(* IEC 61131-3 sources: scada_scout/plc_programs, 162 files *)

(* ---- PRG_GBCUPM01.st ---- *)
(* ========================================================================
   PLC PROGRAM: PRG_GBCUPM01
   IED: GBCUPM01
   Device: GBCUPM01
   Generated: 2026-02-05 10:55:39

   This program runs cyclically (default 100ms) and has access to all
   data points of the associated IEC 61850 device. Users can add custom
   logic in the designated sections below.
   ======================================================================== *)

PROGRAM PRG_GBCUPM01
VAR
    (* ====== System Variables ====== *)
    cycle_count: UDINT := 0;           (* Increments each scan cycle *)
    first_scan: BOOL := TRUE;          (* TRUE only on first execution *)
    scan_time_ms: REAL := 0.0;         (* Last scan time in milliseconds *)

    (* ====== IED Connection Status ====== *)
    ied_connected: BOOL := FALSE;      (* TRUE when IED server is running *)
    ied_name: STRING := 'GBCUPM01';
    device_name: STRING := 'GBCUPM01';

    (* ====== Logical Devices ====== *)
    (* Available LDs: AnUn_ArcProtInput1, Application, BinIO, BinIO_BinaryInputs, BinIO_BinaryOutputs, CB1, CB1_Fundamental, Ds1, Ds2, Mod1, Mod1_Channel1, Mod2, Mod2_Channel1, Mod3, Mod3_Channel1, PowS, PowS_MeasPointI3ph1, PowS_MeasPointV3ph1, Rec, Rec_FaultRecorder, VI3p1, VI3p1_5051NOCgndB1, VI3p1_5051OC3phase1, VI3p1_ArcProtection1, VI3p1_Energy, VI3p1_FundSymComp, VI3p1_OperationalValues, VI3p1_ProcessMonitor, CB2, CB2_Fundamental, CB3, CB3_Fundamental, ComSupervision, ComSupervision_GOOSE *)

    (* ====== User Variables ====== *)
    (* Add your custom variables here *)
    (* Example:
    timer1: TON;
    counter: INT := 0;
    status_word: WORD;
    *)

END_VAR

(* ======================================================================
   INITIALIZATION SECTION
   Runs once on first scan. Use for setup and initialization.
   ====================================================================== *)
IF first_scan THEN
    (* Initialize user variables here *)
    cycle_count := 0;

    (* Log program start *)
    (* SCADA_LOG('INFO', CONCAT('PLC Program started: ', device_name)); *)

    first_scan := FALSE;
END_IF;

(* ======================================================================
   MAIN CYCLIC EXECUTION
   This section runs continuously every scan cycle (default 100ms).
   ====================================================================== *)

(* Increment cycle counter *)
cycle_count := cycle_count + 1;

(* ====== USER LOGIC SECTION 1: Pre-Processing ====== *)
(* Add logic that should run before main processing *)
(* Example:
IF ied_connected THEN
    (* Read IED data points *)
    (* status_word := READ_IED_DATA(device_name, 'LD0/MMXU1$MX$TotW$mag'); *)
END_IF;
*)

(* ====== USER LOGIC SECTION 2: Main Processing ====== *)
(* Add your main control logic here *)
(* Example:
IF counter > 100 THEN
    counter := 0;
    (* Perform periodic action *)
END_IF;
counter := counter + 1;
*)

(* ====== USER LOGIC SECTION 3: Post-Processing ====== *)
(* Add logic for outputs, writes, and cleanup *)
(* Example:
IF ied_connected THEN
    (* Write control commands to IED *)
    (* WRITE_IED_CONTROL(device_name, 'LD0/CSWI1$CO$Pos', TRUE); *)
END_IF;
*)

(* ====== Built-in Functions Available ====== *)
(*
   READ_IED_DATA(device: STRING, ref: STRING): ANY
       - Read data from IED object reference
       - Example: READ_IED_DATA('MyIED', 'LD0/MMXU1$MX$TotW$mag')

   WRITE_IED_DATA(device: STRING, ref: STRING, value: ANY): BOOL
       - Write data to IED object reference
       - Returns TRUE on success

   WRITE_IED_CONTROL(device: STRING, ref: STRING, value: ANY): BOOL
       - Send control command to IED
       - Returns TRUE on success

   SCADA_LOG(level: STRING, message: STRING)
       - Log message to event log
       - Levels: 'INFO', 'WARNING', 'ERROR'

   GET_DEVICE_STATUS(device: STRING): BOOL
       - Check if device is connected
*)

END_PROGRAM

(* ---- PRG_GPS01ECB01.st ---- *)
(* ========================================================================
   PLC PROGRAM: PRG_GPS01ECB01
   IED: GPS01ECB01
   Device: GPS01ECB01
   Generated: 2026-02-05 10:51:13

   This program runs cyclically (default 100ms) and has access to all
   data points of the associated IEC 61850 device. Users can add custom
   logic in the designated sections below.
   ======================================================================== *)

PROGRAM PRG_GPS01ECB01
VAR
    (* ====== System Variables ====== *)
    cycle_count: UDINT := 0;           (* Increments each scan cycle *)
    first_scan: BOOL := TRUE;          (* TRUE only on first execution *)
    scan_time_ms: REAL := 0.0;         (* Last scan time in milliseconds *)

    (* ====== IED Connection Status ====== *)
    ied_connected: BOOL := FALSE;      (* TRUE when IED server is running *)
    ied_name: STRING := 'GPS01ECB01';
    device_name: STRING := 'GPS01ECB01';

    (* ====== Logical Devices ====== *)
    (* Available LDs: AnUn_ArcProtInput1, Application, BinIO, BinIO_BinaryInputs, BinIO_BinaryOutputs, CB1, CB1_Fundamental, Ds1, Ds2, Mod1, Mod1_Channel1, Mod2, Mod2_Channel1, Mod3, Mod3_Channel1, PowS, PowS_MeasPointI3ph1, PowS_MeasPointV3ph1, Rec, Rec_FaultRecorder, VI3p1, VI3p1_5051NOCgndB1, VI3p1_5051OC3phase1, VI3p1_67DirOC3phB1, VI3p1_67NDirOCgndB1, VI3p1_ArcProtection1, VI3p1_Energy, VI3p1_FundSymComp, VI3p1_OperationalValues, VI3p1_ProcessMonitor, VI3p1_ExternalTrip1, VI3p1_ExternalTrip2, PowS_MeasPointI1ph1, VI1p1, VI1p1_50N51NOC1phB1, VI1p1_Fundamental, ComSupervision, ComSupervision_GOOSE *)

    (* ====== User Variables ====== *)
    (* Add your custom variables here *)
    (* Example:
    timer1: TON;
    counter: INT := 0;
    status_word: WORD;
    *)

END_VAR

(* ======================================================================
   INITIALIZATION SECTION
   Runs once on first scan. Use for setup and initialization.
   ====================================================================== *)
IF first_scan THEN
    (* Initialize user variables here *)
    cycle_count := 0;

    (* Log program start *)
    (* SCADA_LOG('INFO', CONCAT('PLC Program started: ', device_name)); *)

    first_scan := FALSE;
END_IF;

(* ======================================================================
   MAIN CYCLIC EXECUTION
   This section runs continuously every scan cycle (default 100ms).
   ====================================================================== *)

(* Increment cycle counter *)
cycle_count := cycle_count + 1;

(* ====== USER LOGIC SECTION 1: Pre-Processing ====== *)
(* Add logic that should run before main processing *)
(* Example:
IF ied_connected THEN
    (* Read IED data points *)
    (* status_word := READ_IED_DATA(device_name, 'LD0/MMXU1$MX$TotW$mag'); *)
END_IF;
*)

(* ====== USER LOGIC SECTION 2: Main Processing ====== *)
(* Add your main control logic here *)
(* Example:
IF counter > 100 THEN
    counter := 0;
    (* Perform periodic action *)
END_IF;
counter := counter + 1;
*)

(* ====== USER LOGIC SECTION 3: Post-Processing ====== *)
(* Add logic for outputs, writes, and cleanup *)
(* Example:
IF ied_connected THEN
    (* Write control commands to IED *)
    (* WRITE_IED_CONTROL(device_name, 'LD0/CSWI1$CO$Pos', TRUE); *)
END_IF;
*)

(* ====== Built-in Functions Available ====== *)
(*
   READ_IED_DATA(device: STRING, ref: STRING): ANY
       - Read data from IED object reference
       - Example: READ_IED_DATA('MyIED', 'LD0/MMXU1$MX$TotW$mag')

   WRITE_IED_DATA(device: STRING, ref: STRING, value: ANY): BOOL
       - Write data to IED object reference
       - Returns TRUE on success

   WRITE_IED_CONTROL(device: STRING, ref: STRING, value: ANY): BOOL
       - Send control command to IED
       - Returns TRUE on success

   SCADA_LOG(level: STRING, message: STRING)
       - Log message to event log
       - Levels: 'INFO', 'WARNING', 'ERROR'

   GET_DEVICE_STATUS(device: STRING): BOOL
       - Check if device is connected
*)

END_PROGRAM

(* ---- PRG_GPS01FCB01.st ---- *)
(* ========================================================================
   PLC PROGRAM: PRG_GPS01FCB01
   IED: GPS01FCB01
   Device: GPS01FCB01
   Generated: 2026-02-05 10:51:08

   This program runs cyclically (default 100ms) and has access to all
   data points of the associated IEC 61850 device. Users can add custom
   logic in the designated sections below.
   ======================================================================== *)

PROGRAM PRG_GPS01FCB01
VAR
    (* ====== System Variables ====== *)
    cycle_count: UDINT := 0;           (* Increments each scan cycle *)
    first_scan: BOOL := TRUE;          (* TRUE only on first execution *)
    scan_time_ms: REAL := 0.0;         (* Last scan time in milliseconds *)

    (* ====== IED Connection Status ====== *)
    ied_connected: BOOL := FALSE;      (* TRUE when IED server is running *)
    ied_name: STRING := 'GPS01FCB01';
    device_name: STRING := 'GPS01FCB01';

    (* ====== Logical Devices ====== *)
    (* Available LDs: AnUn_ArcProtInput1, Application, BinIO, BinIO_BinaryInputs, BinIO_BinaryOutputs, CB1, CB1_Fundamental, Ds1, Ds2, Mod1, Mod1_Channel1, Mod2, Mod2_Channel1, Mod3, Mod3_Channel1, PowS, PowS_MeasPointI3ph1, PowS_MeasPointV1ph1, PowS_MeasPointV3ph1, Rec, Rec_FaultRecorder, VI1p1, VI1p1_Fundamental, VI3p1, VI3p1_5051NOCgndB1, VI3p1_5051OC3phase1, VI3p1_67DirOC3phB1, VI3p1_67NDirOCgndB1, VI3p1_ArcProtection1, VI3p1_Energy, VI3p1_FundSymComp, VI3p1_OperationalValues, VI3p1_ProcessMonitor, VI3p1_ExternalTrip1, VI3p1_ExternalTrip2, ComSupervision, ComSupervision_GOOSE *)

    (* ====== User Variables ====== *)
    (* Add your custom variables here *)
    (* Example:
    timer1: TON;
    counter: INT := 0;
    status_word: WORD;
    *)

END_VAR

(* ======================================================================
   INITIALIZATION SECTION
   Runs once on first scan. Use for setup and initialization.
   ====================================================================== *)
IF first_scan THEN
    (* Initialize user variables here *)
    cycle_count := 0;

    (* Log program start *)
    (* SCADA_LOG('INFO', CONCAT('PLC Program started: ', device_name)); *)

    first_scan := FALSE;
END_IF;

(* ======================================================================
   MAIN CYCLIC EXECUTION
   This section runs continuously every scan cycle (default 100ms).
   ====================================================================== *)

(* Increment cycle counter *)
cycle_count := cycle_count + 1;

(* ====== USER LOGIC SECTION 1: Pre-Processing ====== *)
(* Add logic that should run before main processing *)
(* Example:
IF ied_connected THEN
    (* Read IED data points *)
    (* status_word := READ_IED_DATA(device_name, 'LD0/MMXU1$MX$TotW$mag'); *)
END_IF;
*)

(* ====== USER LOGIC SECTION 2: Main Processing ====== *)
(* Add your main control logic here *)
(* Example:
IF counter > 100 THEN
    counter := 0;
    (* Perform periodic action *)
END_IF;
counter := counter + 1;
*)

(* ====== USER LOGIC SECTION 3: Post-Processing ====== *)
(* Add logic for outputs, writes, and cleanup *)
(* Example:
IF ied_connected THEN
    (* Write control commands to IED *)
    (* WRITE_IED_CONTROL(device_name, 'LD0/CSWI1$CO$Pos', TRUE); *)
END_IF;
*)

(* ====== Built-in Functions Available ====== *)
(*
   READ_IED_DATA(device: STRING, ref: STRING): ANY
       - Read data from IED object reference
       - Example: READ_IED_DATA('MyIED', 'LD0/MMXU1$MX$TotW$mag')

   WRITE_IED_DATA(device: STRING, ref: STRING, value: ANY): BOOL
       - Write data to IED object reference
       - Returns TRUE on success

   WRITE_IED_CONTROL(device: STRING, ref: STRING, value: ANY): BOOL
       - Send control command to IED
       - Returns TRUE on success

   SCADA_LOG(level: STRING, message: STRING)
       - Log message to event log
       - Levels: 'INFO', 'WARNING', 'ERROR'

   GET_DEVICE_STATUS(device: STRING): BOOL
       - Check if device is connected
*)

END_PROGRAM

(* ---- PRG_GPS01FCB02.st ---- *)
(* ========================================================================
   PLC PROGRAM: PRG_GPS01FCB02
   IED: GPS01FCB02
   Device: GPS01FCB02
   Generated: 2026-02-05 10:51:10

   This program runs cyclically (default 100ms) and has access to all
   data points of the associated IEC 61850 device. Users can add custom
   logic in the designated sections below.
   ======================================================================== *)

PROGRAM PRG_GPS01FCB02
VAR
    (* ====== System Variables ====== *)
    cycle_count: UDINT := 0;           (* Increments each scan cycle *)
    first_scan: BOOL := TRUE;          (* TRUE only on first execution *)
    scan_time_ms: REAL := 0.0;         (* Last scan time in milliseconds *)

    (* ====== IED Connection Status ====== *)
    ied_connected: BOOL := FALSE;      (* TRUE when IED server is running *)
    ied_name: STRING := 'GPS01FCB02';
    device_name: STRING := 'GPS01FCB02';

    (* ====== Logical Devices ====== *)
    (* Available LDs: AnUn_ArcProtInput1, Application, BinIO, BinIO_BinaryInputs, BinIO_BinaryOutputs, CB1, CB1_Fundamental, Ds1, Ds2, Mod1, Mod1_Channel1, Mod2, Mod2_Channel1, Mod3, Mod3_Channel1, PowS, PowS_MeasPointI3ph1, PowS_MeasPointV1ph1, PowS_MeasPointV3ph1, Rec, Rec_FaultRecorder, VI1p1, VI1p1_Fundamental, VI3p1, VI3p1_5051NOCgndB1, VI3p1_5051OC3phase1, VI3p1_67DirOC3phB1, VI3p1_67NDirOCgndB1, VI3p1_ArcProtection1, VI3p1_Energy, VI3p1_FundSymComp, VI3p1_OperationalValues, VI3p1_ProcessMonitor, VI3p1_ExternalTrip1, VI3p1_ExternalTrip2, ComSupervision, ComSupervision_GOOSE *)

    (* ====== User Variables ====== *)
    (* Add your custom variables here *)
    (* Example:
    timer1: TON;
    counter: INT := 0;
    status_word: WORD;
    *)

END_VAR

(* ======================================================================
   INITIALIZATION SECTION
   Runs once on first scan. Use for setup and initialization.
   ====================================================================== *)
IF first_scan THEN
    (* Initialize user variables here *)
    cycle_count := 0;

    (* Log program start *)
    (* SCADA_LOG('INFO', CONCAT('PLC Program started: ', device_name)); *)

    first_scan := FALSE;
END_IF;

(* ======================================================================
   MAIN CYCLIC EXECUTION
   This section runs continuously every scan cycle (default 100ms).
   ====================================================================== *)

(* Increment cycle counter *)
cycle_count := cycle_count + 1;

(* ====== USER LOGIC SECTION 1: Pre-Processing ====== *)
(* Add logic that should run before main processing *)
(* Example:
IF ied_connected THEN
    (* Read IED data points *)
    (* status_word := READ_IED_DATA(device_name, 'LD0/MMXU1$MX$TotW$mag'); *)
END_IF;
*)

(* ====== USER LOGIC SECTION 2: Main Processing ====== *)
(* Add your main control logic here *)
(* Example:
IF counter > 100 THEN
    counter := 0;
    (* Perform periodic action *)
END_IF;
counter := counter + 1;
*)

(* ====== USER LOGIC SECTION 3: Post-Processing ====== *)
(* Add logic for outputs, writes, and cleanup *)
(* Example:
IF ied_connected THEN
    (* Write control commands to IED *)
    (* WRITE_IED_CONTROL(device_name, 'LD0/CSWI1$CO$Pos', TRUE); *)
END_IF;
*)

(* ====== Built-in Functions Available ====== *)
(*
   READ_IED_DATA(device: STRING, ref: STRING): ANY
       - Read data from IED object reference
       - Example: READ_IED_DATA('MyIED', 'LD0/MMXU1$MX$TotW$mag')

   WRITE_IED_DATA(device: STRING, ref: STRING, value: ANY): BOOL
       - Write data to IED object reference
       - Returns TRUE on success

   WRITE_IED_CONTROL(device: STRING, ref: STRING, value: ANY): BOOL
       - Send control command to IED
       - Returns TRUE on success

   SCADA_LOG(level: STRING, message: STRING)
       - Log message to event log
       - Levels: 'INFO', 'WARNING', 'ERROR'

   GET_DEVICE_STATUS(device: STRING): BOOL
       - Check if device is connected
*)

END_PROGRAM

(* ---- PRG_GPS01FCB03.st ---- *)
(* ========================================================================
   PLC PROGRAM: PRG_GPS01FCB03
   IED: GPS01FCB03
   Device: GPS01FCB03
   Generated: 2026-02-05 10:51:23

   This program runs cyclically (default 100ms) and has access to all
   data points of the associated IEC 61850 device. Users can add custom
   logic in the designated sections below.
   ======================================================================== *)

PROGRAM PRG_GPS01FCB03
VAR
    (* ====== System Variables ====== *)
    cycle_count: UDINT := 0;           (* Increments each scan cycle *)
    first_scan: BOOL := TRUE;          (* TRUE only on first execution *)
    scan_time_ms: REAL := 0.0;         (* Last scan time in milliseconds *)

    (* ====== IED Connection Status ====== *)
    ied_connected: BOOL := FALSE;      (* TRUE when IED server is running *)
    ied_name: STRING := 'GPS01FCB03';
    device_name: STRING := 'GPS01FCB03';

    (* ====== Logical Devices ====== *)
    (* Available LDs: AnUn_ArcProtInput1, Application, BinIO, BinIO_BinaryInputs, BinIO_BinaryOutputs, CB1, CB1_Fundamental, Ds1, Ds2, Mod1, Mod1_Channel1, Mod2, Mod2_Channel1, Mod3, Mod3_Channel1, PowS, PowS_MeasPointI3ph1, PowS_MeasPointV1ph1, PowS_MeasPointV3ph1, Rec, Rec_FaultRecorder, VI1p1, VI1p1_Fundamental, VI3p1, VI3p1_5051NOCgndB1, VI3p1_5051OC3phase1, VI3p1_67DirOC3phB1, VI3p1_67NDirOCgndB1, VI3p1_ArcProtection1, VI3p1_Energy, VI3p1_FundSymComp, VI3p1_OperationalValues, VI3p1_ProcessMonitor, VI3p1_ExternalTrip1, VI3p1_ExternalTrip2, ComSupervision, ComSupervision_GOOSE *)

    (* ====== User Variables ====== *)
    (* Add your custom variables here *)
    (* Example:
    timer1: TON;
    counter: INT := 0;
    status_word: WORD;
    *)

END_VAR

(* ======================================================================
   INITIALIZATION SECTION
   Runs once on first scan. Use for setup and initialization.
   ====================================================================== *)
IF first_scan THEN
    (* Initialize user variables here *)
    cycle_count := 0;

    (* Log program start *)
    (* SCADA_LOG('INFO', CONCAT('PLC Program started: ', device_name)); *)

    first_scan := FALSE;
END_IF;

(* ======================================================================
   MAIN CYCLIC EXECUTION
   This section runs continuously every scan cycle (default 100ms).
   ====================================================================== *)

(* Increment cycle counter *)
cycle_count := cycle_count + 1;

(* ====== USER LOGIC SECTION 1: Pre-Processing ====== *)
(* Add logic that should run before main processing *)
(* Example:
IF ied_connected THEN
    (* Read IED data points *)
    (* status_word := READ_IED_DATA(device_name, 'LD0/MMXU1$MX$TotW$mag'); *)
END_IF;
*)

(* ====== USER LOGIC SECTION 2: Main Processing ====== *)
(* Add your main control logic here *)
(* Example:
IF counter > 100 THEN
    counter := 0;
    (* Perform periodic action *)
END_IF;
counter := counter + 1;
*)

(* ====== USER LOGIC SECTION 3: Post-Processing ====== *)
(* Add logic for outputs, writes, and cleanup *)
(* Example:
IF ied_connected THEN
    (* Write control commands to IED *)
    (* WRITE_IED_CONTROL(device_name, 'LD0/CSWI1$CO$Pos', TRUE); *)
END_IF;
*)

(* ====== Built-in Functions Available ====== *)
(*
   READ_IED_DATA(device: STRING, ref: STRING): ANY
       - Read data from IED object reference
       - Example: READ_IED_DATA('MyIED', 'LD0/MMXU1$MX$TotW$mag')

   WRITE_IED_DATA(device: STRING, ref: STRING, value: ANY): BOOL
       - Write data to IED object reference
       - Returns TRUE on success

   WRITE_IED_CONTROL(device: STRING, ref: STRING, value: ANY): BOOL
       - Send control command to IED
       - Returns TRUE on success

   SCADA_LOG(level: STRING, message: STRING)
       - Log message to event log
       - Levels: 'INFO', 'WARNING', 'ERROR'

   GET_DEVICE_STATUS(device: STRING): BOOL
       - Check if device is connected
*)

END_PROGRAM

(* ---- PRG_GPS01FCB04.st ---- *)
(* ========================================================================
   PLC PROGRAM: PRG_GPS01FCB04
   IED: GPS01FCB04
   Device: GPS01FCB04
   Generated: 2026-02-05 10:51:16

   This program runs cyclically (default 100ms) and has access to all
   data points of the associated IEC 61850 device. Users can add custom
   logic in the designated sections below.
   ======================================================================== *)

PROGRAM PRG_GPS01FCB04
VAR
    (* ====== System Variables ====== *)
    cycle_count: UDINT := 0;           (* Increments each scan cycle *)
    first_scan: BOOL := TRUE;          (* TRUE only on first execution *)
    scan_time_ms: REAL := 0.0;         (* Last scan time in milliseconds *)

    (* ====== IED Connection Status ====== *)
    ied_connected: BOOL := FALSE;      (* TRUE when IED server is running *)
    ied_name: STRING := 'GPS01FCB04';
    device_name: STRING := 'GPS01FCB04';

    (* ====== Logical Devices ====== *)
    (* Available LDs: AnUn_ArcProtInput1, Application, BinIO, BinIO_BinaryInputs, BinIO_BinaryOutputs, CB1, CB1_Fundamental, Ds1, Ds2, Mod1, Mod1_Channel1, Mod2, Mod2_Channel1, Mod3, Mod3_Channel1, PowS, PowS_MeasPointI3ph1, PowS_MeasPointV1ph1, PowS_MeasPointV3ph1, Rec, Rec_FaultRecorder, VI1p1, VI1p1_Fundamental, VI3p1, VI3p1_5051NOCgndB1, VI3p1_5051OC3phase1, VI3p1_67DirOC3phB1, VI3p1_67NDirOCgndB1, VI3p1_ArcProtection1, VI3p1_Energy, VI3p1_FundSymComp, VI3p1_OperationalValues, VI3p1_ProcessMonitor, VI3p1_ExternalTrip1, VI3p1_ExternalTrip2, VI3p1_ExternalTrip3, ComSupervision, ComSupervision_GOOSE *)

    (* ====== User Variables ====== *)
    (* Add your custom variables here *)
    (* Example:
    timer1: TON;
    counter: INT := 0;
    status_word: WORD;
    *)

END_VAR

(* ======================================================================
   INITIALIZATION SECTION
   Runs once on first scan. Use for setup and initialization.
   ====================================================================== *)
IF first_scan THEN
    (* Initialize user variables here *)
    cycle_count := 0;

    (* Log program start *)
    (* SCADA_LOG('INFO', CONCAT('PLC Program started: ', device_name)); *)

    first_scan := FALSE;
END_IF;

(* ======================================================================
   MAIN CYCLIC EXECUTION
   This section runs continuously every scan cycle (default 100ms).
   ====================================================================== *)

(* Increment cycle counter *)
cycle_count := cycle_count + 1;

(* ====== USER LOGIC SECTION 1: Pre-Processing ====== *)
(* Add logic that should run before main processing *)
(* Example:
IF ied_connected THEN
    (* Read IED data points *)
    (* status_word := READ_IED_DATA(device_name, 'LD0/MMXU1$MX$TotW$mag'); *)
END_IF;
*)

(* ====== USER LOGIC SECTION 2: Main Processing ====== *)
(* Add your main control logic here *)
(* Example:
IF counter > 100 THEN
    counter := 0;
    (* Perform periodic action *)
END_IF;
counter := counter + 1;
*)

(* ====== USER LOGIC SECTION 3: Post-Processing ====== *)
(* Add logic for outputs, writes, and cleanup *)
(* Example:
IF ied_connected THEN
    (* Write control commands to IED *)
    (* WRITE_IED_CONTROL(device_name, 'LD0/CSWI1$CO$Pos', TRUE); *)
END_IF;
*)

(* ====== Built-in Functions Available ====== *)
(*
   READ_IED_DATA(device: STRING, ref: STRING): ANY
       - Read data from IED object reference
       - Example: READ_IED_DATA('MyIED', 'LD0/MMXU1$MX$TotW$mag')

   WRITE_IED_DATA(device: STRING, ref: STRING, value: ANY): BOOL
       - Write data to IED object reference
       - Returns TRUE on success

   WRITE_IED_CONTROL(device: STRING, ref: STRING, value: ANY): BOOL
       - Send control command to IED
       - Returns TRUE on success

   SCADA_LOG(level: STRING, message: STRING)
       - Log message to event log
       - Levels: 'INFO', 'WARNING', 'ERROR'

   GET_DEVICE_STATUS(device: STRING): BOOL
       - Check if device is connected
*)

END_PROGRAM

(* ---- PRG_GPS01FCB05.st ---- *)
(* ========================================================================
   PLC PROGRAM: PRG_GPS01FCB05
   IED: GPS01FCB05
   Device: GPS01FCB05
   Generated: 2026-02-05 10:51:18

   This program runs cyclically (default 100ms) and has access to all
   data points of the associated IEC 61850 device. Users can add custom
   logic in the designated sections below.
   ======================================================================== *)

PROGRAM PRG_GPS01FCB05
VAR
    (* ====== System Variables ====== *)
    cycle_count: UDINT := 0;           (* Increments each scan cycle *)
    first_scan: BOOL := TRUE;          (* TRUE only on first execution *)
    scan_time_ms: REAL := 0.0;         (* Last scan time in milliseconds *)

    (* ====== IED Connection Status ====== *)
    ied_connected: BOOL := FALSE;      (* TRUE when IED server is running *)
    ied_name: STRING := 'GPS01FCB05';
    device_name: STRING := 'GPS01FCB05';

    (* ====== Logical Devices ====== *)
    (* Available LDs: AnUn_ArcProtInput1, Application, BinIO, BinIO_BinaryInputs, BinIO_BinaryOutputs, CB1, CB1_Fundamental, Ds1, Ds2, Mod1, Mod1_Channel1, Mod2, Mod2_Channel1, Mod3, Mod3_Channel1, PowS, PowS_MeasPointI3ph1, PowS_MeasPointV1ph1, PowS_MeasPointV3ph1, Rec, Rec_FaultRecorder, VI1p1, VI1p1_Fundamental, VI3p1, VI3p1_5051NOCgndB1, VI3p1_5051OC3phase1, VI3p1_67DirOC3phB1, VI3p1_67NDirOCgndB1, VI3p1_ArcProtection1, VI3p1_Energy, VI3p1_FundSymComp, VI3p1_OperationalValues, VI3p1_ProcessMonitor, VI3p1_ExternalTrip1, VI3p1_ExternalTrip2, ComSupervision, ComSupervision_GOOSE *)

    (* ====== User Variables ====== *)
    (* Add your custom variables here *)
    (* Example:
    timer1: TON;
    counter: INT := 0;
    status_word: WORD;
    *)

END_VAR

(* ======================================================================
   INITIALIZATION SECTION
   Runs once on first scan. Use for setup and initialization.
   ====================================================================== *)
IF first_scan THEN
    (* Initialize user variables here *)
    cycle_count := 0;

    (* Log program start *)
    (* SCADA_LOG('INFO', CONCAT('PLC Program started: ', device_name)); *)

    first_scan := FALSE;
END_IF;

(* ======================================================================
   MAIN CYCLIC EXECUTION
   This section runs continuously every scan cycle (default 100ms).
   ====================================================================== *)

(* Increment cycle counter *)
cycle_count := cycle_count + 1;

(* ====== USER LOGIC SECTION 1: Pre-Processing ====== *)
(* Add logic that should run before main processing *)
(* Example:
IF ied_connected THEN
    (* Read IED data points *)
    (* status_word := READ_IED_DATA(device_name, 'LD0/MMXU1$MX$TotW$mag'); *)
END_IF;
*)

(* ====== USER LOGIC SECTION 2: Main Processing ====== *)
(* Add your main control logic here *)
(* Example:
IF counter > 100 THEN
    counter := 0;
    (* Perform periodic action *)
END_IF;
counter := counter + 1;
*)

(* ====== USER LOGIC SECTION 3: Post-Processing ====== *)
(* Add logic for outputs, writes, and cleanup *)
(* Example:
IF ied_connected THEN
    (* Write control commands to IED *)
    (* WRITE_IED_CONTROL(device_name, 'LD0/CSWI1$CO$Pos', TRUE); *)
END_IF;
*)

(* ====== Built-in Functions Available ====== *)
(*
   READ_IED_DATA(device: STRING, ref: STRING): ANY
       - Read data from IED object reference
       - Example: READ_IED_DATA('MyIED', 'LD0/MMXU1$MX$TotW$mag')

   WRITE_IED_DATA(device: STRING, ref: STRING, value: ANY): BOOL
       - Write data to IED object reference
       - Returns TRUE on success

   WRITE_IED_CONTROL(device: STRING, ref: STRING, value: ANY): BOOL
       - Send control command to IED
       - Returns TRUE on success

   SCADA_LOG(level: STRING, message: STRING)
       - Log message to event log
       - Levels: 'INFO', 'WARNING', 'ERROR'

   GET_DEVICE_STATUS(device: STRING): BOOL
       - Check if device is connected
*)

END_PROGRAM

(* ---- PRG_GPS01GCB01.st ---- *)
(* ========================================================================
   PLC PROGRAM: PRG_GPS01GCB01
   IED: GPS01GCB01
   Device: GPS01GCB01
   Generated: 2026-02-05 10:50:31

   This program runs cyclically (default 100ms) and has access to all
   data points of the associated IEC 61850 device. Users can add custom
   logic in the designated sections below.
   ======================================================================== *)

PROGRAM PRG_GPS01GCB01
VAR
    (* ====== System Variables ====== *)
    cycle_count: UDINT := 0;           (* Increments each scan cycle *)
    first_scan: BOOL := TRUE;          (* TRUE only on first execution *)
    scan_time_ms: REAL := 0.0;         (* Last scan time in milliseconds *)

    (* ====== IED Connection Status ====== *)
    ied_connected: BOOL := FALSE;      (* TRUE when IED server is running *)
    ied_name: STRING := 'GPS01GCB01';
    device_name: STRING := 'GPS01GCB01';

    (* ====== Logical Devices ====== *)
    (* Available LDs: AnUn_ArcProtInput1, Application, BinIO, BinIO_BinaryInputs, BinIO_BinaryOutputs, CB1, CB1_25Synchronization, CB1_Fundamental, Ds1, Ds2, Mod1, Mod1_Channel1, Mod2, Mod2_Channel1, Mod3, Mod3_Channel1, PowS, PowS_MeasPointI3ph1, PowS_MeasPointV1ph1, PowS_MeasPointV3ph1, Rec, Rec_FaultRecorder, VI1p1, VI1p1_Fundamental, VI3p1, VI3p1_5051NOCgndB1, VI3p1_5051OC3phase1, VI3p1_67DirOC3phB1, VI3p1_67NDirOCgndB1, VI3p1_ArcProtection1, VI3p1_Energy, VI3p1_FundSymComp, VI3p1_OperationalValues, VI3p1_ProcessMonitor, VI3p1_ExternalTrip1, VI3p1_ExternalTrip2, ComSupervision, ComSupervision_GOOSE *)

    (* ====== User Variables ====== *)
    (* Add your custom variables here *)
    (* Example:
    timer1: TON;
    counter: INT := 0;
    status_word: WORD;
    *)

END_VAR

(* ======================================================================
   INITIALIZATION SECTION
   Runs once on first scan. Use for setup and initialization.
   ====================================================================== *)
IF first_scan THEN
    (* Initialize user variables here *)
    cycle_count := 0;

    (* Log program start *)
    (* SCADA_LOG('INFO', CONCAT('PLC Program started: ', device_name)); *)

    first_scan := FALSE;
END_IF;

(* ======================================================================
   MAIN CYCLIC EXECUTION
   This section runs continuously every scan cycle (default 100ms).
   ====================================================================== *)

(* Increment cycle counter *)
cycle_count := cycle_count + 1;

(* ====== USER LOGIC SECTION 1: Pre-Processing ====== *)
(* Add logic that should run before main processing *)
(* Example:
IF ied_connected THEN
    (* Read IED data points *)
    (* status_word := READ_IED_DATA(device_name, 'LD0/MMXU1$MX$TotW$mag'); *)
END_IF;
*)

(* ====== USER LOGIC SECTION 2: Main Processing ====== *)
(* Add your main control logic here *)
(* Example:
IF counter > 100 THEN
    counter := 0;
    (* Perform periodic action *)
END_IF;
counter := counter + 1;
*)

(* ====== USER LOGIC SECTION 3: Post-Processing ====== *)
(* Add logic for outputs, writes, and cleanup *)
(* Example:
IF ied_connected THEN
    (* Write control commands to IED *)
    (* WRITE_IED_CONTROL(device_name, 'LD0/CSWI1$CO$Pos', TRUE); *)
END_IF;
*)

(* ====== Built-in Functions Available ====== *)
(*
   READ_IED_DATA(device: STRING, ref: STRING): ANY
       - Read data from IED object reference
       - Example: READ_IED_DATA('MyIED', 'LD0/MMXU1$MX$TotW$mag')

   WRITE_IED_DATA(device: STRING, ref: STRING, value: ANY): BOOL
       - Write data to IED object reference
       - Returns TRUE on success

   WRITE_IED_CONTROL(device: STRING, ref: STRING, value: ANY): BOOL
       - Send control command to IED
       - Returns TRUE on success

   SCADA_LOG(level: STRING, message: STRING)
       - Log message to event log
       - Levels: 'INFO', 'WARNING', 'ERROR'

   GET_DEVICE_STATUS(device: STRING): BOOL
       - Check if device is connected
*)

END_PROGRAM

(* ---- PRG_GPS01GCB02.st ---- *)
(* ========================================================================
   PLC PROGRAM: PRG_GPS01GCB02
   IED: GPS01GCB02
   Device: GPS01GCB02
   Generated: 2026-02-05 10:50:36

   This program runs cyclically (default 100ms) and has access to all
   data points of the associated IEC 61850 device. Users can add custom
   logic in the designated sections below.
   ======================================================================== *)

PROGRAM PRG_GPS01GCB02
VAR
    (* ====== System Variables ====== *)
    cycle_count: UDINT := 0;           (* Increments each scan cycle *)
    first_scan: BOOL := TRUE;          (* TRUE only on first execution *)
    scan_time_ms: REAL := 0.0;         (* Last scan time in milliseconds *)

    (* ====== IED Connection Status ====== *)
    ied_connected: BOOL := FALSE;      (* TRUE when IED server is running *)
    ied_name: STRING := 'GPS01GCB02';
    device_name: STRING := 'GPS01GCB02';

    (* ====== Logical Devices ====== *)
    (* Available LDs: AnUn_ArcProtInput1, Application, BinIO, BinIO_BinaryInputs, BinIO_BinaryOutputs, CB1, CB1_25Synchronization, CB1_Fundamental, Ds1, Ds2, Mod1, Mod1_Channel1, Mod2, Mod2_Channel1, Mod3, Mod3_Channel1, PowS, PowS_MeasPointI3ph1, PowS_MeasPointV1ph1, PowS_MeasPointV3ph1, Rec, Rec_FaultRecorder, VI1p1, VI1p1_Fundamental, VI3p1, VI3p1_5051NOCgndB1, VI3p1_5051OC3phase1, VI3p1_67DirOC3phB1, VI3p1_67NDirOCgndB1, VI3p1_ArcProtection1, VI3p1_Energy, VI3p1_FundSymComp, VI3p1_OperationalValues, VI3p1_ProcessMonitor, VI3p1_ExternalTrip1, VI3p1_ExternalTrip2, ComSupervision, ComSupervision_GOOSE *)

    (* ====== User Variables ====== *)
    (* Add your custom variables here *)
    (* Example:
    timer1: TON;
    counter: INT := 0;
    status_word: WORD;
    *)

END_VAR

(* ======================================================================
   INITIALIZATION SECTION
   Runs once on first scan. Use for setup and initialization.
   ====================================================================== *)
IF first_scan THEN
    (* Initialize user variables here *)
    cycle_count := 0;

    (* Log program start *)
    (* SCADA_LOG('INFO', CONCAT('PLC Program started: ', device_name)); *)

    first_scan := FALSE;
END_IF;

(* ======================================================================
   MAIN CYCLIC EXECUTION
   This section runs continuously every scan cycle (default 100ms).
   ====================================================================== *)

(* Increment cycle counter *)
cycle_count := cycle_count + 1;

(* ====== USER LOGIC SECTION 1: Pre-Processing ====== *)
(* Add logic that should run before main processing *)
(* Example:
IF ied_connected THEN
    (* Read IED data points *)
    (* status_word := READ_IED_DATA(device_name, 'LD0/MMXU1$MX$TotW$mag'); *)
END_IF;
*)

(* ====== USER LOGIC SECTION 2: Main Processing ====== *)
(* Add your main control logic here *)
(* Example:
IF counter > 100 THEN
    counter := 0;
    (* Perform periodic action *)
END_IF;
counter := counter + 1;
*)

(* ====== USER LOGIC SECTION 3: Post-Processing ====== *)
(* Add logic for outputs, writes, and cleanup *)
(* Example:
IF ied_connected THEN
    (* Write control commands to IED *)
    (* WRITE_IED_CONTROL(device_name, 'LD0/CSWI1$CO$Pos', TRUE); *)
END_IF;
*)

(* ====== Built-in Functions Available ====== *)
(*
   READ_IED_DATA(device: STRING, ref: STRING): ANY
       - Read data from IED object reference
       - Example: READ_IED_DATA('MyIED', 'LD0/MMXU1$MX$TotW$mag')

   WRITE_IED_DATA(device: STRING, ref: STRING, value: ANY): BOOL
       - Write data to IED object reference
       - Returns TRUE on success

   WRITE_IED_CONTROL(device: STRING, ref: STRING, value: ANY): BOOL
       - Send control command to IED
       - Returns TRUE on success

   SCADA_LOG(level: STRING, message: STRING)
       - Log message to event log
       - Levels: 'INFO', 'WARNING', 'ERROR'

   GET_DEVICE_STATUS(device: STRING): BOOL
       - Check if device is connected
*)

END_PROGRAM

(* ---- PRG_GPS01GCB03.st ---- *)
(* ========================================================================
   PLC PROGRAM: PRG_GPS01GCB03
   IED: GPS01GCB03
   Device: GPS01GCB03
   Generated: 2026-02-05 10:50:41

   This program runs cyclically (default 100ms) and has access to all
   data points of the associated IEC 61850 device. Users can add custom
   logic in the designated sections below.
   ======================================================================== *)

PROGRAM PRG_GPS01GCB03
VAR
    (* ====== System Variables ====== *)
    cycle_count: UDINT := 0;           (* Increments each scan cycle *)
    first_scan: BOOL := TRUE;          (* TRUE only on first execution *)
    scan_time_ms: REAL := 0.0;         (* Last scan time in milliseconds *)

    (* ====== IED Connection Status ====== *)
    ied_connected: BOOL := FALSE;      (* TRUE when IED server is running *)
    ied_name: STRING := 'GPS01GCB03';
    device_name: STRING := 'GPS01GCB03';

    (* ====== Logical Devices ====== *)
    (* Available LDs: AnUn_ArcProtInput1, Application, BinIO, BinIO_BinaryInputs, BinIO_BinaryOutputs, CB1, CB1_25Synchronization, CB1_Fundamental, Ds1, Ds2, Mod1, Mod1_Channel1, Mod2, Mod2_Channel1, Mod3, Mod3_Channel1, PowS, PowS_MeasPointI3ph1, PowS_MeasPointV1ph1, PowS_MeasPointV3ph1, Rec, Rec_FaultRecorder, VI1p1, VI1p1_Fundamental, VI3p1, VI3p1_5051NOCgndB1, VI3p1_5051OC3phase1, VI3p1_67DirOC3phB1, VI3p1_67NDirOCgndB1, VI3p1_ArcProtection1, VI3p1_Energy, VI3p1_FundSymComp, VI3p1_OperationalValues, VI3p1_ProcessMonitor, VI3p1_ExternalTrip1, VI3p1_ExternalTrip2, ComSupervision, ComSupervision_GOOSE *)

    (* ====== User Variables ====== *)
    (* Add your custom variables here *)
    (* Example:
    timer1: TON;
    counter: INT := 0;
    status_word: WORD;
    *)

END_VAR

(* ======================================================================
   INITIALIZATION SECTION
   Runs once on first scan. Use for setup and initialization.
   ====================================================================== *)
IF first_scan THEN
    (* Initialize user variables here *)
    cycle_count := 0;

    (* Log program start *)
    (* SCADA_LOG('INFO', CONCAT('PLC Program started: ', device_name)); *)

    first_scan := FALSE;
END_IF;

(* ======================================================================
   MAIN CYCLIC EXECUTION
   This section runs continuously every scan cycle (default 100ms).
   ====================================================================== *)

(* Increment cycle counter *)
cycle_count := cycle_count + 1;

(* ====== USER LOGIC SECTION 1: Pre-Processing ====== *)
(* Add logic that should run before main processing *)
(* Example:
IF ied_connected THEN
    (* Read IED data points *)
    (* status_word := READ_IED_DATA(device_name, 'LD0/MMXU1$MX$TotW$mag'); *)
END_IF;
*)

(* ====== USER LOGIC SECTION 2: Main Processing ====== *)
(* Add your main control logic here *)
(* Example:
IF counter > 100 THEN
    counter := 0;
    (* Perform periodic action *)
END_IF;
counter := counter + 1;
*)

(* ====== USER LOGIC SECTION 3: Post-Processing ====== *)
(* Add logic for outputs, writes, and cleanup *)
(* Example:
IF ied_connected THEN
    (* Write control commands to IED *)
    (* WRITE_IED_CONTROL(device_name, 'LD0/CSWI1$CO$Pos', TRUE); *)
END_IF;
*)

(* ====== Built-in Functions Available ====== *)
(*
   READ_IED_DATA(device: STRING, ref: STRING): ANY
       - Read data from IED object reference
       - Example: READ_IED_DATA('MyIED', 'LD0/MMXU1$MX$TotW$mag')

   WRITE_IED_DATA(device: STRING, ref: STRING, value: ANY): BOOL
       - Write data to IED object reference
       - Returns TRUE on success

   WRITE_IED_CONTROL(device: STRING, ref: STRING, value: ANY): BOOL
       - Send control command to IED
       - Returns TRUE on success

   SCADA_LOG(level: STRING, message: STRING)
       - Log message to event log
       - Levels: 'INFO', 'WARNING', 'ERROR'

   GET_DEVICE_STATUS(device: STRING): BOOL
       - Check if device is connected
*)

END_PROGRAM

(* ---- PRG_GPS01GCB04.st ---- *)
(* ========================================================================
   PLC PROGRAM: PRG_GPS01GCB04
   IED: GPS01GCB04
   Device: GPS01GCB04
   Generated: 2026-02-05 10:50:52

   This program runs cyclically (default 100ms) and has access to all
   data points of the associated IEC 61850 device. Users can add custom
   logic in the designated sections below.
   ======================================================================== *)

PROGRAM PRG_GPS01GCB04
VAR
    (* ====== System Variables ====== *)
    cycle_count: UDINT := 0;           (* Increments each scan cycle *)
    first_scan: BOOL := TRUE;          (* TRUE only on first execution *)
    scan_time_ms: REAL := 0.0;         (* Last scan time in milliseconds *)

    (* ====== IED Connection Status ====== *)
    ied_connected: BOOL := FALSE;      (* TRUE when IED server is running *)
    ied_name: STRING := 'GPS01GCB04';
    device_name: STRING := 'GPS01GCB04';

    (* ====== Logical Devices ====== *)
    (* Available LDs: AnUn_ArcProtInput1, Application, BinIO, BinIO_BinaryInputs, BinIO_BinaryOutputs, CB1, CB1_25Synchronization, CB1_Fundamental, Ds1, Ds2, Mod1, Mod1_Channel1, Mod2, Mod2_Channel1, Mod3, Mod3_Channel1, PowS, PowS_MeasPointI3ph1, PowS_MeasPointV1ph1, PowS_MeasPointV3ph1, Rec, Rec_FaultRecorder, VI1p1, VI1p1_Fundamental, VI3p1, VI3p1_5051NOCgndB1, VI3p1_5051OC3phase1, VI3p1_67DirOC3phB1, VI3p1_67NDirOCgndB1, VI3p1_ArcProtection1, VI3p1_Energy, VI3p1_FundSymComp, VI3p1_OperationalValues, VI3p1_ProcessMonitor, VI3p1_ExternalTrip1, VI3p1_ExternalTrip2, ComSupervision, ComSupervision_GOOSE *)

    (* ====== User Variables ====== *)
    (* Add your custom variables here *)
    (* Example:
    timer1: TON;
    counter: INT := 0;
    status_word: WORD;
    *)

END_VAR

(* ======================================================================
   INITIALIZATION SECTION
   Runs once on first scan. Use for setup and initialization.
   ====================================================================== *)
IF first_scan THEN
    (* Initialize user variables here *)
    cycle_count := 0;

    (* Log program start *)
    (* SCADA_LOG('INFO', CONCAT('PLC Program started: ', device_name)); *)

    first_scan := FALSE;
END_IF;

(* ======================================================================
   MAIN CYCLIC EXECUTION
   This section runs continuously every scan cycle (default 100ms).
   ====================================================================== *)

(* Increment cycle counter *)
cycle_count := cycle_count + 1;

(* ====== USER LOGIC SECTION 1: Pre-Processing ====== *)
(* Add logic that should run before main processing *)
(* Example:
IF ied_connected THEN
    (* Read IED data points *)
    (* status_word := READ_IED_DATA(device_name, 'LD0/MMXU1$MX$TotW$mag'); *)
END_IF;
*)

(* ====== USER LOGIC SECTION 2: Main Processing ====== *)
(* Add your main control logic here *)
(* Example:
IF counter > 100 THEN
    counter := 0;
    (* Perform periodic action *)
END_IF;
counter := counter + 1;
*)

(* ====== USER LOGIC SECTION 3: Post-Processing ====== *)
(* Add logic for outputs, writes, and cleanup *)
(* Example:
IF ied_connected THEN
    (* Write control commands to IED *)
    (* WRITE_IED_CONTROL(device_name, 'LD0/CSWI1$CO$Pos', TRUE); *)
END_IF;
*)

(* ====== Built-in Functions Available ====== *)
(*
   READ_IED_DATA(device: STRING, ref: STRING): ANY
       - Read data from IED object reference
       - Example: READ_IED_DATA('MyIED', 'LD0/MMXU1$MX$TotW$mag')

   WRITE_IED_DATA(device: STRING, ref: STRING, value: ANY): BOOL
       - Write data to IED object reference
       - Returns TRUE on success

   WRITE_IED_CONTROL(device: STRING, ref: STRING, value: ANY): BOOL
       - Send control command to IED
       - Returns TRUE on success

   SCADA_LOG(level: STRING, message: STRING)
       - Log message to event log
       - Levels: 'INFO', 'WARNING', 'ERROR'

   GET_DEVICE_STATUS(device: STRING): BOOL
       - Check if device is connected
*)

END_PROGRAM

(* ---- PRG_GPS01GCB05.st ---- *)
(* ========================================================================
   PLC PROGRAM: PRG_GPS01GCB05
   IED: GPS01GCB05
   Device: GPS01GCB05
   Generated: 2026-02-05 10:50:56

   This program runs cyclically (default 100ms) and has access to all
   data points of the associated IEC 61850 device. Users can add custom
   logic in the designated sections below.
   ======================================================================== *)

PROGRAM PRG_GPS01GCB05
VAR
    (* ====== System Variables ====== *)
    cycle_count: UDINT := 0;           (* Increments each scan cycle *)
    first_scan: BOOL := TRUE;          (* TRUE only on first execution *)
    scan_time_ms: REAL := 0.0;         (* Last scan time in milliseconds *)

    (* ====== IED Connection Status ====== *)
    ied_connected: BOOL := FALSE;      (* TRUE when IED server is running *)
    ied_name: STRING := 'GPS01GCB05';
    device_name: STRING := 'GPS01GCB05';

    (* ====== Logical Devices ====== *)
    (* Available LDs: AnUn_ArcProtInput1, Application, BinIO, BinIO_BinaryInputs, BinIO_BinaryOutputs, CB1, CB1_25Synchronization, CB1_Fundamental, Ds1, Ds2, Mod1, Mod1_Channel1, Mod2, Mod2_Channel1, Mod3, Mod3_Channel1, PowS, PowS_MeasPointI3ph1, PowS_MeasPointV1ph1, PowS_MeasPointV3ph1, Rec, Rec_FaultRecorder, VI1p1, VI1p1_Fundamental, VI3p1, VI3p1_5051NOCgndB1, VI3p1_5051OC3phase1, VI3p1_67DirOC3phB1, VI3p1_67NDirOCgndB1, VI3p1_ArcProtection1, VI3p1_Energy, VI3p1_FundSymComp, VI3p1_OperationalValues, VI3p1_ProcessMonitor, VI3p1_ExternalTrip1, VI3p1_ExternalTrip2, ComSupervision, ComSupervision_GOOSE *)

    (* ====== User Variables ====== *)
    (* Add your custom variables here *)
    (* Example:
    timer1: TON;
    counter: INT := 0;
    status_word: WORD;
    *)

END_VAR

(* ======================================================================
   INITIALIZATION SECTION
   Runs once on first scan. Use for setup and initialization.
   ====================================================================== *)
IF first_scan THEN
    (* Initialize user variables here *)
    cycle_count := 0;

    (* Log program start *)
    (* SCADA_LOG('INFO', CONCAT('PLC Program started: ', device_name)); *)

    first_scan := FALSE;
END_IF;

(* ======================================================================
   MAIN CYCLIC EXECUTION
   This section runs continuously every scan cycle (default 100ms).
   ====================================================================== *)

(* Increment cycle counter *)
cycle_count := cycle_count + 1;

(* ====== USER LOGIC SECTION 1: Pre-Processing ====== *)
(* Add logic that should run before main processing *)
(* Example:
IF ied_connected THEN
    (* Read IED data points *)
    (* status_word := READ_IED_DATA(device_name, 'LD0/MMXU1$MX$TotW$mag'); *)
END_IF;
*)

(* ====== USER LOGIC SECTION 2: Main Processing ====== *)
(* Add your main control logic here *)
(* Example:
IF counter > 100 THEN
    counter := 0;
    (* Perform periodic action *)
END_IF;
counter := counter + 1;
*)

(* ====== USER LOGIC SECTION 3: Post-Processing ====== *)
(* Add logic for outputs, writes, and cleanup *)
(* Example:
IF ied_connected THEN
    (* Write control commands to IED *)
    (* WRITE_IED_CONTROL(device_name, 'LD0/CSWI1$CO$Pos', TRUE); *)
END_IF;
*)

(* ====== Built-in Functions Available ====== *)
(*
   READ_IED_DATA(device: STRING, ref: STRING): ANY
       - Read data from IED object reference
       - Example: READ_IED_DATA('MyIED', 'LD0/MMXU1$MX$TotW$mag')

   WRITE_IED_DATA(device: STRING, ref: STRING, value: ANY): BOOL
       - Write data to IED object reference
       - Returns TRUE on success

   WRITE_IED_CONTROL(device: STRING, ref: STRING, value: ANY): BOOL
       - Send control command to IED
       - Returns TRUE on success

   SCADA_LOG(level: STRING, message: STRING)
       - Log message to event log
       - Levels: 'INFO', 'WARNING', 'ERROR'

   GET_DEVICE_STATUS(device: STRING): BOOL
       - Check if device is connected
*)

END_PROGRAM

(* ---- PRG_GPS01GCB06.st ---- *)
(* ========================================================================
   PLC PROGRAM: PRG_GPS01GCB06
   IED: GPS01GCB06
   Device: GPS01GCB06
   Generated: 2026-02-05 10:51:01

   This program runs cyclically (default 100ms) and has access to all
   data points of the associated IEC 61850 device. Users can add custom
   logic in the designated sections below.
   ======================================================================== *)

PROGRAM PRG_GPS01GCB06
VAR
    (* ====== System Variables ====== *)
    cycle_count: UDINT := 0;           (* Increments each scan cycle *)
    first_scan: BOOL := TRUE;          (* TRUE only on first execution *)
    scan_time_ms: REAL := 0.0;         (* Last scan time in milliseconds *)

    (* ====== IED Connection Status ====== *)
    ied_connected: BOOL := FALSE;      (* TRUE when IED server is running *)
    ied_name: STRING := 'GPS01GCB06';
    device_name: STRING := 'GPS01GCB06';

    (* ====== Logical Devices ====== *)
    (* Available LDs: AnUn_ArcProtInput1, Application, BinIO, BinIO_BinaryInputs, BinIO_BinaryOutputs, CB1, CB1_25Synchronization, CB1_Fundamental, Ds1, Ds2, Mod1, Mod1_Channel1, Mod2, Mod2_Channel1, Mod3, Mod3_Channel1, PowS, PowS_MeasPointI3ph1, PowS_MeasPointV1ph1, PowS_MeasPointV3ph1, Rec, Rec_FaultRecorder, VI1p1, VI1p1_Fundamental, VI3p1, VI3p1_5051NOCgndB1, VI3p1_5051OC3phase1, VI3p1_67DirOC3phB1, VI3p1_67NDirOCgndB1, VI3p1_ArcProtection1, VI3p1_Energy, VI3p1_FundSymComp, VI3p1_OperationalValues, VI3p1_ProcessMonitor, VI3p1_ExternalTrip1, VI3p1_ExternalTrip2, ComSupervision, ComSupervision_GOOSE *)

    (* ====== User Variables ====== *)
    (* Add your custom variables here *)
    (* Example:
    timer1: TON;
    counter: INT := 0;
    status_word: WORD;
    *)

END_VAR

(* ======================================================================
   INITIALIZATION SECTION
   Runs once on first scan. Use for setup and initialization.
   ====================================================================== *)
IF first_scan THEN
    (* Initialize user variables here *)
    cycle_count := 0;

    (* Log program start *)
    (* SCADA_LOG('INFO', CONCAT('PLC Program started: ', device_name)); *)

    first_scan := FALSE;
END_IF;

(* ======================================================================
   MAIN CYCLIC EXECUTION
   This section runs continuously every scan cycle (default 100ms).
   ====================================================================== *)

(* Increment cycle counter *)
cycle_count := cycle_count + 1;

(* ====== USER LOGIC SECTION 1: Pre-Processing ====== *)
(* Add logic that should run before main processing *)
(* Example:
IF ied_connected THEN
    (* Read IED data points *)
    (* status_word := READ_IED_DATA(device_name, 'LD0/MMXU1$MX$TotW$mag'); *)
END_IF;
*)

(* ====== USER LOGIC SECTION 2: Main Processing ====== *)
(* Add your main control logic here *)
(* Example:
IF counter > 100 THEN
    counter := 0;
    (* Perform periodic action *)
END_IF;
counter := counter + 1;
*)

(* ====== USER LOGIC SECTION 3: Post-Processing ====== *)
(* Add logic for outputs, writes, and cleanup *)
(* Example:
IF ied_connected THEN
    (* Write control commands to IED *)
    (* WRITE_IED_CONTROL(device_name, 'LD0/CSWI1$CO$Pos', TRUE); *)
END_IF;
*)

(* ====== Built-in Functions Available ====== *)
(*
   READ_IED_DATA(device: STRING, ref: STRING): ANY
       - Read data from IED object reference
       - Example: READ_IED_DATA('MyIED', 'LD0/MMXU1$MX$TotW$mag')

   WRITE_IED_DATA(device: STRING, ref: STRING, value: ANY): BOOL
       - Write data to IED object reference
       - Returns TRUE on success

   WRITE_IED_CONTROL(device: STRING, ref: STRING, value: ANY): BOOL
       - Send control command to IED
       - Returns TRUE on success

   SCADA_LOG(level: STRING, message: STRING)
       - Log message to event log
       - Levels: 'INFO', 'WARNING', 'ERROR'

   GET_DEVICE_STATUS(device: STRING): BOOL
       - Check if device is connected
*)

END_PROGRAM

(* ---- PRG_GPS01GCB07.st ---- *)
(* ========================================================================
   PLC PROGRAM: PRG_GPS01GCB07
   IED: GPS01GCB07
   Device: GPS01GCB07
   Generated: 2026-02-05 10:51:06

   This program runs cyclically (default 100ms) and has access to all
   data points of the associated IEC 61850 device. Users can add custom
   logic in the designated sections below.
   ======================================================================== *)

PROGRAM PRG_GPS01GCB07
VAR
    (* ====== System Variables ====== *)
    cycle_count: UDINT := 0;           (* Increments each scan cycle *)
    first_scan: BOOL := TRUE;          (* TRUE only on first execution *)
    scan_time_ms: REAL := 0.0;         (* Last scan time in milliseconds *)

    (* ====== IED Connection Status ====== *)
    ied_connected: BOOL := FALSE;      (* TRUE when IED server is running *)
    ied_name: STRING := 'GPS01GCB07';
    device_name: STRING := 'GPS01GCB07';

    (* ====== Logical Devices ====== *)
    (* Available LDs: AnUn_ArcProtInput1, Application, BinIO, BinIO_BinaryInputs, BinIO_BinaryOutputs, CB1, CB1_25Synchronization, CB1_Fundamental, Ds1, Ds2, Mod1, Mod1_Channel1, Mod2, Mod2_Channel1, Mod3, Mod3_Channel1, PowS, PowS_MeasPointI3ph1, PowS_MeasPointV1ph1, PowS_MeasPointV3ph1, Rec, Rec_FaultRecorder, VI1p1, VI1p1_Fundamental, VI3p1, VI3p1_5051NOCgndB1, VI3p1_5051OC3phase1, VI3p1_67DirOC3phB1, VI3p1_67NDirOCgndB1, VI3p1_ArcProtection1, VI3p1_Energy, VI3p1_FundSymComp, VI3p1_OperationalValues, VI3p1_ProcessMonitor, VI3p1_ExternalTrip1, VI3p1_ExternalTrip2, ComSupervision, ComSupervision_GOOSE *)

    (* ====== User Variables ====== *)
    (* Add your custom variables here *)
    (* Example:
    timer1: TON;
    counter: INT := 0;
    status_word: WORD;
    *)

END_VAR

(* ======================================================================
   INITIALIZATION SECTION
   Runs once on first scan. Use for setup and initialization.
   ====================================================================== *)
IF first_scan THEN
    (* Initialize user variables here *)
    cycle_count := 0;

    (* Log program start *)
    (* SCADA_LOG('INFO', CONCAT('PLC Program started: ', device_name)); *)

    first_scan := FALSE;
END_IF;

(* ======================================================================
   MAIN CYCLIC EXECUTION
   This section runs continuously every scan cycle (default 100ms).
   ====================================================================== *)

(* Increment cycle counter *)
cycle_count := cycle_count + 1;

(* ====== USER LOGIC SECTION 1: Pre-Processing ====== *)
(* Add logic that should run before main processing *)
(* Example:
IF ied_connected THEN
    (* Read IED data points *)
    (* status_word := READ_IED_DATA(device_name, 'LD0/MMXU1$MX$TotW$mag'); *)
END_IF;
*)

(* ====== USER LOGIC SECTION 2: Main Processing ====== *)
(* Add your main control logic here *)
(* Example:
IF counter > 100 THEN
    counter := 0;
    (* Perform periodic action *)
END_IF;
counter := counter + 1;
*)

(* ====== USER LOGIC SECTION 3: Post-Processing ====== *)
(* Add logic for outputs, writes, and cleanup *)
(* Example:
IF ied_connected THEN
    (* Write control commands to IED *)
    (* WRITE_IED_CONTROL(device_name, 'LD0/CSWI1$CO$Pos', TRUE); *)
END_IF;
*)

(* ====== Built-in Functions Available ====== *)
(*
   READ_IED_DATA(device: STRING, ref: STRING): ANY
       - Read data from IED object reference
       - Example: READ_IED_DATA('MyIED', 'LD0/MMXU1$MX$TotW$mag')

   WRITE_IED_DATA(device: STRING, ref: STRING, value: ANY): BOOL
       - Write data to IED object reference
       - Returns TRUE on success

   WRITE_IED_CONTROL(device: STRING, ref: STRING, value: ANY): BOOL
       - Send control command to IED
       - Returns TRUE on success

   SCADA_LOG(level: STRING, message: STRING)
       - Log message to event log
       - Levels: 'INFO', 'WARNING', 'ERROR'

   GET_DEVICE_STATUS(device: STRING): BOOL
       - Check if device is connected
*)

END_PROGRAM

(* ---- PRG_GPS01GCB08.st ---- *)
(* ========================================================================
   PLC PROGRAM: PRG_GPS01GCB08
   IED: GPS01GCB08
   Device: GPS01GCB08
   Generated: 2026-02-05 10:50:32

   This program runs cyclically (default 100ms) and has access to all
   data points of the associated IEC 61850 device. Users can add custom
   logic in the designated sections below.
   ======================================================================== *)

PROGRAM PRG_GPS01GCB08
VAR
    (* ====== System Variables ====== *)
    cycle_count: UDINT := 0;           (* Increments each scan cycle *)
    first_scan: BOOL := TRUE;          (* TRUE only on first execution *)
    scan_time_ms: REAL := 0.0;         (* Last scan time in milliseconds *)

    (* ====== IED Connection Status ====== *)
    ied_connected: BOOL := FALSE;      (* TRUE when IED server is running *)
    ied_name: STRING := 'GPS01GCB08';
    device_name: STRING := 'GPS01GCB08';

    (* ====== Logical Devices ====== *)
    (* Available LDs: AnUn_ArcProtInput1, Application, BinIO, BinIO_BinaryInputs, BinIO_BinaryOutputs, CB1, CB1_25Synchronization, CB1_Fundamental, Ds1, Ds2, Mod1, Mod1_Channel1, Mod2, Mod2_Channel1, Mod3, Mod3_Channel1, PowS, PowS_MeasPointI3ph1, PowS_MeasPointV1ph1, PowS_MeasPointV3ph1, Rec, Rec_FaultRecorder, VI1p1, VI1p1_Fundamental, VI3p1, VI3p1_5051NOCgndB1, VI3p1_5051OC3phase1, VI3p1_67DirOC3phB1, VI3p1_67NDirOCgndB1, VI3p1_ArcProtection1, VI3p1_Energy, VI3p1_FundSymComp, VI3p1_OperationalValues, VI3p1_ProcessMonitor, VI3p1_ExternalTrip1, VI3p1_ExternalTrip2, ComSupervision, ComSupervision_GOOSE *)

    (* ====== User Variables ====== *)
    (* Add your custom variables here *)
    (* Example:
    timer1: TON;
    counter: INT := 0;
    status_word: WORD;
    *)

END_VAR

(* ======================================================================
   INITIALIZATION SECTION
   Runs once on first scan. Use for setup and initialization.
   ====================================================================== *)
IF first_scan THEN
    (* Initialize user variables here *)
    cycle_count := 0;

    (* Log program start *)
    (* SCADA_LOG('INFO', CONCAT('PLC Program started: ', device_name)); *)

    first_scan := FALSE;
END_IF;

(* ======================================================================
   MAIN CYCLIC EXECUTION
   This section runs continuously every scan cycle (default 100ms).
   ====================================================================== *)

(* Increment cycle counter *)
cycle_count := cycle_count + 1;

(* ====== USER LOGIC SECTION 1: Pre-Processing ====== *)
(* Add logic that should run before main processing *)
(* Example:
IF ied_connected THEN
    (* Read IED data points *)
    (* status_word := READ_IED_DATA(device_name, 'LD0/MMXU1$MX$TotW$mag'); *)
END_IF;
*)

(* ====== USER LOGIC SECTION 2: Main Processing ====== *)
(* Add your main control logic here *)
(* Example:
IF counter > 100 THEN
    counter := 0;
    (* Perform periodic action *)
END_IF;
counter := counter + 1;
*)

(* ====== USER LOGIC SECTION 3: Post-Processing ====== *)
(* Add logic for outputs, writes, and cleanup *)
(* Example:
IF ied_connected THEN
    (* Write control commands to IED *)
    (* WRITE_IED_CONTROL(device_name, 'LD0/CSWI1$CO$Pos', TRUE); *)
END_IF;
*)

(* ====== Built-in Functions Available ====== *)
(*
   READ_IED_DATA(device: STRING, ref: STRING): ANY
       - Read data from IED object reference
       - Example: READ_IED_DATA('MyIED', 'LD0/MMXU1$MX$TotW$mag')

   WRITE_IED_DATA(device: STRING, ref: STRING, value: ANY): BOOL
       - Write data to IED object reference
       - Returns TRUE on success

   WRITE_IED_CONTROL(device: STRING, ref: STRING, value: ANY): BOOL
       - Send control command to IED
       - Returns TRUE on success

   SCADA_LOG(level: STRING, message: STRING)
       - Log message to event log
       - Levels: 'INFO', 'WARNING', 'ERROR'

   GET_DEVICE_STATUS(device: STRING): BOOL
       - Check if device is connected
*)

END_PROGRAM

(* ---- PRG_GPS01GCB09.st ---- *)
(* ========================================================================
   PLC PROGRAM: PRG_GPS01GCB09
   IED: GPS01GCB09
   Device: GPS01GCB09
   Generated: 2026-02-05 10:50:39

   This program runs cyclically (default 100ms) and has access to all
   data points of the associated IEC 61850 device. Users can add custom
   logic in the designated sections below.
   ======================================================================== *)

PROGRAM PRG_GPS01GCB09
VAR
    (* ====== System Variables ====== *)
    cycle_count: UDINT := 0;           (* Increments each scan cycle *)
    first_scan: BOOL := TRUE;          (* TRUE only on first execution *)
    scan_time_ms: REAL := 0.0;         (* Last scan time in milliseconds *)

    (* ====== IED Connection Status ====== *)
    ied_connected: BOOL := FALSE;      (* TRUE when IED server is running *)
    ied_name: STRING := 'GPS01GCB09';
    device_name: STRING := 'GPS01GCB09';

    (* ====== Logical Devices ====== *)
    (* Available LDs: AnUn_ArcProtInput1, Application, BinIO, BinIO_BinaryInputs, BinIO_BinaryOutputs, CB1, CB1_25Synchronization, CB1_Fundamental, Ds1, Ds2, Mod1, Mod1_Channel1, Mod2, Mod2_Channel1, Mod3, Mod3_Channel1, PowS, PowS_MeasPointI3ph1, PowS_MeasPointV1ph1, PowS_MeasPointV3ph1, Rec, Rec_FaultRecorder, VI1p1, VI1p1_Fundamental, VI3p1, VI3p1_5051NOCgndB1, VI3p1_5051OC3phase1, VI3p1_67DirOC3phB1, VI3p1_67NDirOCgndB1, VI3p1_ArcProtection1, VI3p1_Energy, VI3p1_FundSymComp, VI3p1_OperationalValues, VI3p1_ProcessMonitor, VI3p1_ExternalTrip1, VI3p1_ExternalTrip2, ComSupervision, ComSupervision_GOOSE *)

    (* ====== User Variables ====== *)
    (* Add your custom variables here *)
    (* Example:
    timer1: TON;
    counter: INT := 0;
    status_word: WORD;
    *)

END_VAR

(* ======================================================================
   INITIALIZATION SECTION
   Runs once on first scan. Use for setup and initialization.
   ====================================================================== *)
IF first_scan THEN
    (* Initialize user variables here *)
    cycle_count := 0;

    (* Log program start *)
    (* SCADA_LOG('INFO', CONCAT('PLC Program started: ', device_name)); *)

    first_scan := FALSE;
END_IF;

(* ======================================================================
   MAIN CYCLIC EXECUTION
   This section runs continuously every scan cycle (default 100ms).
   ====================================================================== *)

(* Increment cycle counter *)
cycle_count := cycle_count + 1;

(* ====== USER LOGIC SECTION 1: Pre-Processing ====== *)
(* Add logic that should run before main processing *)
(* Example:
IF ied_connected THEN
    (* Read IED data points *)
    (* status_word := READ_IED_DATA(device_name, 'LD0/MMXU1$MX$TotW$mag'); *)
END_IF;
*)

(* ====== USER LOGIC SECTION 2: Main Processing ====== *)
(* Add your main control logic here *)
(* Example:
IF counter > 100 THEN
    counter := 0;
    (* Perform periodic action *)
END_IF;
counter := counter + 1;
*)

(* ====== USER LOGIC SECTION 3: Post-Processing ====== *)
(* Add logic for outputs, writes, and cleanup *)
(* Example:
IF ied_connected THEN
    (* Write control commands to IED *)
    (* WRITE_IED_CONTROL(device_name, 'LD0/CSWI1$CO$Pos', TRUE); *)
END_IF;
*)

(* ====== Built-in Functions Available ====== *)
(*
   READ_IED_DATA(device: STRING, ref: STRING): ANY
       - Read data from IED object reference
       - Example: READ_IED_DATA('MyIED', 'LD0/MMXU1$MX$TotW$mag')

   WRITE_IED_DATA(device: STRING, ref: STRING, value: ANY): BOOL
       - Write data to IED object reference
       - Returns TRUE on success

   WRITE_IED_CONTROL(device: STRING, ref: STRING, value: ANY): BOOL
       - Send control command to IED
       - Returns TRUE on success

   SCADA_LOG(level: STRING, message: STRING)
       - Log message to event log
       - Levels: 'INFO', 'WARNING', 'ERROR'

   GET_DEVICE_STATUS(device: STRING): BOOL
       - Check if device is connected
*)

END_PROGRAM

(* ---- PRG_GPS01GCB10.st ---- *)
(* ========================================================================
   PLC PROGRAM: PRG_GPS01GCB10
   IED: GPS01GCB10
   Device: GPS01GCB10
   Generated: 2026-02-05 10:50:45

   This program runs cyclically (default 100ms) and has access to all
   data points of the associated IEC 61850 device. Users can add custom
   logic in the designated sections below.
   ======================================================================== *)

PROGRAM PRG_GPS01GCB10
VAR
    (* ====== System Variables ====== *)
    cycle_count: UDINT := 0;           (* Increments each scan cycle *)
    first_scan: BOOL := TRUE;          (* TRUE only on first execution *)
    scan_time_ms: REAL := 0.0;         (* Last scan time in milliseconds *)

    (* ====== IED Connection Status ====== *)
    ied_connected: BOOL := FALSE;      (* TRUE when IED server is running *)
    ied_name: STRING := 'GPS01GCB10';
    device_name: STRING := 'GPS01GCB10';

    (* ====== Logical Devices ====== *)
    (* Available LDs: AnUn_ArcProtInput1, Application, BinIO, BinIO_BinaryInputs, BinIO_BinaryOutputs, CB1, CB1_25Synchronization, CB1_Fundamental, Ds1, Ds2, Mod1, Mod1_Channel1, Mod2, Mod2_Channel1, Mod3, Mod3_Channel1, PowS, PowS_MeasPointI3ph1, PowS_MeasPointV1ph1, PowS_MeasPointV3ph1, Rec, Rec_FaultRecorder, VI1p1, VI1p1_Fundamental, VI3p1, VI3p1_5051NOCgndB1, VI3p1_5051OC3phase1, VI3p1_67DirOC3phB1, VI3p1_67NDirOCgndB1, VI3p1_ArcProtection1, VI3p1_Energy, VI3p1_FundSymComp, VI3p1_OperationalValues, VI3p1_ProcessMonitor, VI3p1_ExternalTrip1, VI3p1_ExternalTrip2, ComSupervision, ComSupervision_GOOSE *)

    (* ====== User Variables ====== *)
    (* Add your custom variables here *)
    (* Example:
    timer1: TON;
    counter: INT := 0;
    status_word: WORD;
    *)

END_VAR

(* ======================================================================
   INITIALIZATION SECTION
   Runs once on first scan. Use for setup and initialization.
   ====================================================================== *)
IF first_scan THEN
    (* Initialize user variables here *)
    cycle_count := 0;

    (* Log program start *)
    (* SCADA_LOG('INFO', CONCAT('PLC Program started: ', device_name)); *)

    first_scan := FALSE;
END_IF;

(* ======================================================================
   MAIN CYCLIC EXECUTION
   This section runs continuously every scan cycle (default 100ms).
   ====================================================================== *)

(* Increment cycle counter *)
cycle_count := cycle_count + 1;

(* ====== USER LOGIC SECTION 1: Pre-Processing ====== *)
(* Add logic that should run before main processing *)
(* Example:
IF ied_connected THEN
    (* Read IED data points *)
    (* status_word := READ_IED_DATA(device_name, 'LD0/MMXU1$MX$TotW$mag'); *)
END_IF;
*)

(* ====== USER LOGIC SECTION 2: Main Processing ====== *)
(* Add your main control logic here *)
(* Example:
IF counter > 100 THEN
    counter := 0;
    (* Perform periodic action *)
END_IF;
counter := counter + 1;
*)

(* ====== USER LOGIC SECTION 3: Post-Processing ====== *)
(* Add logic for outputs, writes, and cleanup *)
(* Example:
IF ied_connected THEN
    (* Write control commands to IED *)
    (* WRITE_IED_CONTROL(device_name, 'LD0/CSWI1$CO$Pos', TRUE); *)
END_IF;
*)

(* ====== Built-in Functions Available ====== *)
(*
   READ_IED_DATA(device: STRING, ref: STRING): ANY
       - Read data from IED object reference
       - Example: READ_IED_DATA('MyIED', 'LD0/MMXU1$MX$TotW$mag')

   WRITE_IED_DATA(device: STRING, ref: STRING, value: ANY): BOOL
       - Write data to IED object reference
       - Returns TRUE on success

   WRITE_IED_CONTROL(device: STRING, ref: STRING, value: ANY): BOOL
       - Send control command to IED
       - Returns TRUE on success

   SCADA_LOG(level: STRING, message: STRING)
       - Log message to event log
       - Levels: 'INFO', 'WARNING', 'ERROR'

   GET_DEVICE_STATUS(device: STRING): BOOL
       - Check if device is connected
*)

END_PROGRAM

(* ---- PRG_GPS01GCB11.st ---- *)
(* ========================================================================
   PLC PROGRAM: PRG_GPS01GCB11
   IED: GPS01GCB11
   Device: GPS01GCB11
   Generated: 2026-02-05 10:50:54

   This program runs cyclically (default 100ms) and has access to all
   data points of the associated IEC 61850 device. Users can add custom
   logic in the designated sections below.
   ======================================================================== *)

PROGRAM PRG_GPS01GCB11
VAR
    (* ====== System Variables ====== *)
    cycle_count: UDINT := 0;           (* Increments each scan cycle *)
    first_scan: BOOL := TRUE;          (* TRUE only on first execution *)
    scan_time_ms: REAL := 0.0;         (* Last scan time in milliseconds *)

    (* ====== IED Connection Status ====== *)
    ied_connected: BOOL := FALSE;      (* TRUE when IED server is running *)
    ied_name: STRING := 'GPS01GCB11';
    device_name: STRING := 'GPS01GCB11';

    (* ====== Logical Devices ====== *)
    (* Available LDs: AnUn_ArcProtInput1, Application, BinIO, BinIO_BinaryInputs, BinIO_BinaryOutputs, CB1, CB1_25Synchronization, CB1_Fundamental, Ds1, Ds2, Mod1, Mod1_Channel1, Mod2, Mod2_Channel1, Mod3, Mod3_Channel1, PowS, PowS_MeasPointI3ph1, PowS_MeasPointV1ph1, PowS_MeasPointV3ph1, Rec, Rec_FaultRecorder, VI1p1, VI1p1_Fundamental, VI3p1, VI3p1_5051NOCgndB1, VI3p1_5051OC3phase1, VI3p1_67DirOC3phB1, VI3p1_67NDirOCgndB1, VI3p1_ArcProtection1, VI3p1_Energy, VI3p1_FundSymComp, VI3p1_OperationalValues, VI3p1_ProcessMonitor, VI3p1_ExternalTrip1, VI3p1_ExternalTrip2, ComSupervision, ComSupervision_GOOSE *)

    (* ====== User Variables ====== *)
    (* Add your custom variables here *)
    (* Example:
    timer1: TON;
    counter: INT := 0;
    status_word: WORD;
    *)

END_VAR

(* ======================================================================
   INITIALIZATION SECTION
   Runs once on first scan. Use for setup and initialization.
   ====================================================================== *)
IF first_scan THEN
    (* Initialize user variables here *)
    cycle_count := 0;

    (* Log program start *)
    (* SCADA_LOG('INFO', CONCAT('PLC Program started: ', device_name)); *)

    first_scan := FALSE;
END_IF;

(* ======================================================================
   MAIN CYCLIC EXECUTION
   This section runs continuously every scan cycle (default 100ms).
   ====================================================================== *)

(* Increment cycle counter *)
cycle_count := cycle_count + 1;

(* ====== USER LOGIC SECTION 1: Pre-Processing ====== *)
(* Add logic that should run before main processing *)
(* Example:
IF ied_connected THEN
    (* Read IED data points *)
    (* status_word := READ_IED_DATA(device_name, 'LD0/MMXU1$MX$TotW$mag'); *)
END_IF;
*)

(* ====== USER LOGIC SECTION 2: Main Processing ====== *)
(* Add your main control logic here *)
(* Example:
IF counter > 100 THEN
    counter := 0;
    (* Perform periodic action *)
END_IF;
counter := counter + 1;
*)

(* ====== USER LOGIC SECTION 3: Post-Processing ====== *)
(* Add logic for outputs, writes, and cleanup *)
(* Example:
IF ied_connected THEN
    (* Write control commands to IED *)
    (* WRITE_IED_CONTROL(device_name, 'LD0/CSWI1$CO$Pos', TRUE); *)
END_IF;
*)

(* ====== Built-in Functions Available ====== *)
(*
   READ_IED_DATA(device: STRING, ref: STRING): ANY
       - Read data from IED object reference
       - Example: READ_IED_DATA('MyIED', 'LD0/MMXU1$MX$TotW$mag')

   WRITE_IED_DATA(device: STRING, ref: STRING, value: ANY): BOOL
       - Write data to IED object reference
       - Returns TRUE on success

   WRITE_IED_CONTROL(device: STRING, ref: STRING, value: ANY): BOOL
       - Send control command to IED
       - Returns TRUE on success

   SCADA_LOG(level: STRING, message: STRING)
       - Log message to event log
       - Levels: 'INFO', 'WARNING', 'ERROR'

   GET_DEVICE_STATUS(device: STRING): BOOL
       - Check if device is connected
*)

END_PROGRAM

(* ---- PRG_GPS01GCB12.st ---- *)
(* ========================================================================
   PLC PROGRAM: PRG_GPS01GCB12
   IED: GPS01GCB12
   Device: GPS01GCB12
   Generated: 2026-02-05 10:50:57

   This program runs cyclically (default 100ms) and has access to all
   data points of the associated IEC 61850 device. Users can add custom
   logic in the designated sections below.
   ======================================================================== *)

PROGRAM PRG_GPS01GCB12
VAR
    (* ====== System Variables ====== *)
    cycle_count: UDINT := 0;           (* Increments each scan cycle *)
    first_scan: BOOL := TRUE;          (* TRUE only on first execution *)
    scan_time_ms: REAL := 0.0;         (* Last scan time in milliseconds *)

    (* ====== IED Connection Status ====== *)
    ied_connected: BOOL := FALSE;      (* TRUE when IED server is running *)
    ied_name: STRING := 'GPS01GCB12';
    device_name: STRING := 'GPS01GCB12';

    (* ====== Logical Devices ====== *)
    (* Available LDs: AnUn_ArcProtInput1, Application, BinIO, BinIO_BinaryInputs, BinIO_BinaryOutputs, CB1, CB1_25Synchronization, CB1_Fundamental, Ds1, Ds2, Mod1, Mod1_Channel1, Mod2, Mod2_Channel1, Mod3, Mod3_Channel1, PowS, PowS_MeasPointI3ph1, PowS_MeasPointV1ph1, PowS_MeasPointV3ph1, Rec, Rec_FaultRecorder, VI1p1, VI1p1_Fundamental, VI3p1, VI3p1_5051NOCgndB1, VI3p1_5051OC3phase1, VI3p1_67DirOC3phB1, VI3p1_67NDirOCgndB1, VI3p1_ArcProtection1, VI3p1_Energy, VI3p1_FundSymComp, VI3p1_OperationalValues, VI3p1_ProcessMonitor, VI3p1_ExternalTrip1, VI3p1_ExternalTrip2, ComSupervision, ComSupervision_GOOSE *)

    (* ====== User Variables ====== *)
    (* Add your custom variables here *)
    (* Example:
    timer1: TON;
    counter: INT := 0;
    status_word: WORD;
    *)

END_VAR

(* ======================================================================
   INITIALIZATION SECTION
   Runs once on first scan. Use for setup and initialization.
   ====================================================================== *)
IF first_scan THEN
    (* Initialize user variables here *)
    cycle_count := 0;

    (* Log program start *)
    (* SCADA_LOG('INFO', CONCAT('PLC Program started: ', device_name)); *)

    first_scan := FALSE;
END_IF;

(* ======================================================================
   MAIN CYCLIC EXECUTION
   This section runs continuously every scan cycle (default 100ms).
   ====================================================================== *)

(* Increment cycle counter *)
cycle_count := cycle_count + 1;

(* ====== USER LOGIC SECTION 1: Pre-Processing ====== *)
(* Add logic that should run before main processing *)
(* Example:
IF ied_connected THEN
    (* Read IED data points *)
    (* status_word := READ_IED_DATA(device_name, 'LD0/MMXU1$MX$TotW$mag'); *)
END_IF;
*)

(* ====== USER LOGIC SECTION 2: Main Processing ====== *)
(* Add your main control logic here *)
(* Example:
IF counter > 100 THEN
    counter := 0;
    (* Perform periodic action *)
END_IF;
counter := counter + 1;
*)

(* ====== USER LOGIC SECTION 3: Post-Processing ====== *)
(* Add logic for outputs, writes, and cleanup *)
(* Example:
IF ied_connected THEN
    (* Write control commands to IED *)
    (* WRITE_IED_CONTROL(device_name, 'LD0/CSWI1$CO$Pos', TRUE); *)
END_IF;
*)

(* ====== Built-in Functions Available ====== *)
(*
   READ_IED_DATA(device: STRING, ref: STRING): ANY
       - Read data from IED object reference
       - Example: READ_IED_DATA('MyIED', 'LD0/MMXU1$MX$TotW$mag')

   WRITE_IED_DATA(device: STRING, ref: STRING, value: ANY): BOOL
       - Write data to IED object reference
       - Returns TRUE on success

   WRITE_IED_CONTROL(device: STRING, ref: STRING, value: ANY): BOOL
       - Send control command to IED
       - Returns TRUE on success

   SCADA_LOG(level: STRING, message: STRING)
       - Log message to event log
       - Levels: 'INFO', 'WARNING', 'ERROR'

   GET_DEVICE_STATUS(device: STRING): BOOL
       - Check if device is connected
*)

END_PROGRAM

(* ---- PRG_GPS01GPC01UPM01FCB01.st ---- *)
(* ========================================================================
   PLC PROGRAM: PRG_GPS01GPC01UPM01FCB01
   IED: GPS01GPC01UPM01FCB01
   Device: GPS01GPC01UPM01FCB01
   Generated: 2026-02-05 10:47:32

   This program runs cyclically (default 100ms) and has access to all
   data points of the associated IEC 61850 device. Users can add custom
   logic in the designated sections below.
   ======================================================================== *)

PROGRAM PRG_GPS01GPC01UPM01FCB01
VAR
    (* ====== System Variables ====== *)
    cycle_count: UDINT := 0;           (* Increments each scan cycle *)
    first_scan: BOOL := TRUE;          (* TRUE only on first execution *)
    scan_time_ms: REAL := 0.0;         (* Last scan time in milliseconds *)

    (* ====== IED Connection Status ====== *)
    ied_connected: BOOL := FALSE;      (* TRUE when IED server is running *)
    ied_name: STRING := 'GPS01GPC01UPM01FCB01';
    device_name: STRING := 'GPS01GPC01UPM01FCB01';

    (* ====== Logical Devices ====== *)
    (* Available LDs: AnUn_ArcProtInput1, Application, BinIO, BinIO_BinaryInputs, BinIO_BinaryOutputs, CB1, CB1_Fundamental, Ds1, Ds2, Mod1, Mod1_Channel1, Mod2, Mod2_Channel1, Mod3, Mod3_Channel1, PowS, PowS_MeasPointI3ph1, PowS_MeasPointV3ph1, Rec, Rec_FaultRecorder, VI3p1, VI3p1_5051NOCgndB1, VI3p1_5051OC3phase1, VI3p1_ArcProtection1, VI3p1_Energy, VI3p1_FundSymComp, VI3p1_OperationalValues, VI3p1_ProcessMonitor, VI3p1_ExternalTrip1, VI3p1_67DirOC3phB1, VI3p1_67NDirOCgndB1, ComSupervision, ComSupervision_GOOSE *)

    (* ====== User Variables ====== *)
    (* Add your custom variables here *)
    (* Example:
    timer1: TON;
    counter: INT := 0;
    status_word: WORD;
    *)

END_VAR

(* ======================================================================
   INITIALIZATION SECTION
   Runs once on first scan. Use for setup and initialization.
   ====================================================================== *)
IF first_scan THEN
    (* Initialize user variables here *)
    cycle_count := 0;

    (* Log program start *)
    (* SCADA_LOG('INFO', CONCAT('PLC Program started: ', device_name)); *)

    first_scan := FALSE;
END_IF;

(* ======================================================================
   MAIN CYCLIC EXECUTION
   This section runs continuously every scan cycle (default 100ms).
   ====================================================================== *)

(* Increment cycle counter *)
cycle_count := cycle_count + 1;

(* ====== USER LOGIC SECTION 1: Pre-Processing ====== *)
(* Add logic that should run before main processing *)
(* Example:
IF ied_connected THEN
    (* Read IED data points *)
    (* status_word := READ_IED_DATA(device_name, 'LD0/MMXU1$MX$TotW$mag'); *)
END_IF;
*)

(* ====== USER LOGIC SECTION 2: Main Processing ====== *)
(* Add your main control logic here *)
(* Example:
IF counter > 100 THEN
    counter := 0;
    (* Perform periodic action *)
END_IF;
counter := counter + 1;
*)

(* ====== USER LOGIC SECTION 3: Post-Processing ====== *)
(* Add logic for outputs, writes, and cleanup *)
(* Example:
IF ied_connected THEN
    (* Write control commands to IED *)
    (* WRITE_IED_CONTROL(device_name, 'LD0/CSWI1$CO$Pos', TRUE); *)
END_IF;
*)

(* ====== Built-in Functions Available ====== *)
(*
   READ_IED_DATA(device: STRING, ref: STRING): ANY
       - Read data from IED object reference
       - Example: READ_IED_DATA('MyIED', 'LD0/MMXU1$MX$TotW$mag')

   WRITE_IED_DATA(device: STRING, ref: STRING, value: ANY): BOOL
       - Write data to IED object reference
       - Returns TRUE on success

   WRITE_IED_CONTROL(device: STRING, ref: STRING, value: ANY): BOOL
       - Send control command to IED
       - Returns TRUE on success

   SCADA_LOG(level: STRING, message: STRING)
       - Log message to event log
       - Levels: 'INFO', 'WARNING', 'ERROR'

   GET_DEVICE_STATUS(device: STRING): BOOL
       - Check if device is connected
*)

END_PROGRAM

(* ---- PRG_GPS01GPC01UPM01FCB02.st ---- *)
(* ========================================================================
   PLC PROGRAM: PRG_GPS01GPC01UPM01FCB02
   IED: GPS01GPC01UPM01FCB02
   Device: GPS01GPC01UPM01FCB02
   Generated: 2026-02-05 10:47:32

   This program runs cyclically (default 100ms) and has access to all
   data points of the associated IEC 61850 device. Users can add custom
   logic in the designated sections below.
   ======================================================================== *)

PROGRAM PRG_GPS01GPC01UPM01FCB02
VAR
    (* ====== System Variables ====== *)
    cycle_count: UDINT := 0;           (* Increments each scan cycle *)
    first_scan: BOOL := TRUE;          (* TRUE only on first execution *)
    scan_time_ms: REAL := 0.0;         (* Last scan time in milliseconds *)

    (* ====== IED Connection Status ====== *)
    ied_connected: BOOL := FALSE;      (* TRUE when IED server is running *)
    ied_name: STRING := 'GPS01GPC01UPM01FCB02';
    device_name: STRING := 'GPS01GPC01UPM01FCB02';

    (* ====== Logical Devices ====== *)
    (* Available LDs: AnUn_ArcProtInput1, Application, BinIO, BinIO_BinaryInputs, BinIO_BinaryOutputs, CB1, CB1_Fundamental, Ds1, Ds2, Mod1, Mod1_Channel1, Mod2, Mod2_Channel1, Mod3, Mod3_Channel1, PowS, PowS_MeasPointI3ph1, PowS_MeasPointV3ph1, Rec, Rec_FaultRecorder, VI3p1, VI3p1_5051NOCgndB1, VI3p1_5051OC3phase1, VI3p1_ArcProtection1, VI3p1_Energy, VI3p1_FundSymComp, VI3p1_OperationalValues, VI3p1_ProcessMonitor, VI3p1_ExternalTrip1, VI3p1_67DirOC3phB1, VI3p1_67NDirOCgndB1, ComSupervision, ComSupervision_GOOSE *)

    (* ====== User Variables ====== *)
    (* Add your custom variables here *)
    (* Example:
    timer1: TON;
    counter: INT := 0;
    status_word: WORD;
    *)

END_VAR

(* ======================================================================
   INITIALIZATION SECTION
   Runs once on first scan. Use for setup and initialization.
   ====================================================================== *)
IF first_scan THEN
    (* Initialize user variables here *)
    cycle_count := 0;

    (* Log program start *)
    (* SCADA_LOG('INFO', CONCAT('PLC Program started: ', device_name)); *)

    first_scan := FALSE;
END_IF;

(* ======================================================================
   MAIN CYCLIC EXECUTION
   This section runs continuously every scan cycle (default 100ms).
   ====================================================================== *)

(* Increment cycle counter *)
cycle_count := cycle_count + 1;

(* ====== USER LOGIC SECTION 1: Pre-Processing ====== *)
(* Add logic that should run before main processing *)
(* Example:
IF ied_connected THEN
    (* Read IED data points *)
    (* status_word := READ_IED_DATA(device_name, 'LD0/MMXU1$MX$TotW$mag'); *)
END_IF;
*)

(* ====== USER LOGIC SECTION 2: Main Processing ====== *)
(* Add your main control logic here *)
(* Example:
IF counter > 100 THEN
    counter := 0;
    (* Perform periodic action *)
END_IF;
counter := counter + 1;
*)

(* ====== USER LOGIC SECTION 3: Post-Processing ====== *)
(* Add logic for outputs, writes, and cleanup *)
(* Example:
IF ied_connected THEN
    (* Write control commands to IED *)
    (* WRITE_IED_CONTROL(device_name, 'LD0/CSWI1$CO$Pos', TRUE); *)
END_IF;
*)

(* ====== Built-in Functions Available ====== *)
(*
   READ_IED_DATA(device: STRING, ref: STRING): ANY
       - Read data from IED object reference
       - Example: READ_IED_DATA('MyIED', 'LD0/MMXU1$MX$TotW$mag')

   WRITE_IED_DATA(device: STRING, ref: STRING, value: ANY): BOOL
       - Write data to IED object reference
       - Returns TRUE on success

   WRITE_IED_CONTROL(device: STRING, ref: STRING, value: ANY): BOOL
       - Send control command to IED
       - Returns TRUE on success

   SCADA_LOG(level: STRING, message: STRING)
       - Log message to event log
       - Levels: 'INFO', 'WARNING', 'ERROR'

   GET_DEVICE_STATUS(device: STRING): BOOL
       - Check if device is connected
*)

END_PROGRAM

(* ---- PRG_GPS01GPC01UPM01MCB01.st ---- *)
(* ========================================================================
   PLC PROGRAM: PRG_GPS01GPC01UPM01MCB01
   IED: GPS01GPC01UPM01MCB01
   Device: GPS01GPC01UPM01MCB01
   Generated: 2026-02-05 10:47:32

   This program runs cyclically (default 100ms) and has access to all
   data points of the associated IEC 61850 device. Users can add custom
   logic in the designated sections below.
   ======================================================================== *)

PROGRAM PRG_GPS01GPC01UPM01MCB01
VAR
    (* ====== System Variables ====== *)
    cycle_count: UDINT := 0;           (* Increments each scan cycle *)
    first_scan: BOOL := TRUE;          (* TRUE only on first execution *)
    scan_time_ms: REAL := 0.0;         (* Last scan time in milliseconds *)

    (* ====== IED Connection Status ====== *)
    ied_connected: BOOL := FALSE;      (* TRUE when IED server is running *)
    ied_name: STRING := 'GPS01GPC01UPM01MCB01';
    device_name: STRING := 'GPS01GPC01UPM01MCB01';

    (* ====== Logical Devices ====== *)
    (* Available LDs: AnUn_ArcProtInput1, Application, BinIO, BinIO_BinaryInputs, BinIO_BinaryOutputs, CB1, CB1_Fundamental, Ds1, Ds2, Mod1, Mod1_Channel1, Mod2, Mod2_Channel1, Mod3, Mod3_Channel1, PowS, PowS_MeasPointI3ph1, PowS_MeasPointV3ph1, Rec, Rec_FaultRecorder, VI3p1, VI3p1_5051NOCgndB1, VI3p1_5051OC3phase1, VI3p1_ArcProtection1, VI3p1_Energy, VI3p1_FundSymComp, VI3p1_OperationalValues, VI3p1_ProcessMonitor, VI3p1_ExternalTrip1, VI3p1_67DirOC3phB1, VI3p1_67NDirOCgndB1, VI3p1_ExternalTrip2, ComSupervision, ComSupervision_GOOSE *)

    (* ====== User Variables ====== *)
    (* Add your custom variables here *)
    (* Example:
    timer1: TON;
    counter: INT := 0;
    status_word: WORD;
    *)

END_VAR

(* ======================================================================
   INITIALIZATION SECTION
   Runs once on first scan. Use for setup and initialization.
   ====================================================================== *)
IF first_scan THEN
    (* Initialize user variables here *)
    cycle_count := 0;

    (* Log program start *)
    (* SCADA_LOG('INFO', CONCAT('PLC Program started: ', device_name)); *)

    first_scan := FALSE;
END_IF;

(* ======================================================================
   MAIN CYCLIC EXECUTION
   This section runs continuously every scan cycle (default 100ms).
   ====================================================================== *)

(* Increment cycle counter *)
cycle_count := cycle_count + 1;

(* ====== USER LOGIC SECTION 1: Pre-Processing ====== *)
(* Add logic that should run before main processing *)
(* Example:
IF ied_connected THEN
    (* Read IED data points *)
    (* status_word := READ_IED_DATA(device_name, 'LD0/MMXU1$MX$TotW$mag'); *)
END_IF;
*)

(* ====== USER LOGIC SECTION 2: Main Processing ====== *)
(* Add your main control logic here *)
(* Example:
IF counter > 100 THEN
    counter := 0;
    (* Perform periodic action *)
END_IF;
counter := counter + 1;
*)

(* ====== USER LOGIC SECTION 3: Post-Processing ====== *)
(* Add logic for outputs, writes, and cleanup *)
(* Example:
IF ied_connected THEN
    (* Write control commands to IED *)
    (* WRITE_IED_CONTROL(device_name, 'LD0/CSWI1$CO$Pos', TRUE); *)
END_IF;
*)

(* ====== Built-in Functions Available ====== *)
(*
   READ_IED_DATA(device: STRING, ref: STRING): ANY
       - Read data from IED object reference
       - Example: READ_IED_DATA('MyIED', 'LD0/MMXU1$MX$TotW$mag')

   WRITE_IED_DATA(device: STRING, ref: STRING, value: ANY): BOOL
       - Write data to IED object reference
       - Returns TRUE on success

   WRITE_IED_CONTROL(device: STRING, ref: STRING, value: ANY): BOOL
       - Send control command to IED
       - Returns TRUE on success

   SCADA_LOG(level: STRING, message: STRING)
       - Log message to event log
       - Levels: 'INFO', 'WARNING', 'ERROR'

   GET_DEVICE_STATUS(device: STRING): BOOL
       - Check if device is connected
*)

END_PROGRAM

(* ---- PRG_GPS01GPC02UPM01FCB01.st ---- *)
(* ========================================================================
   PLC PROGRAM: PRG_GPS01GPC02UPM01FCB01
   IED: GPS01GPC02UPM01FCB01
   Device: GPS01GPC02UPM01FCB01
   Generated: 2026-02-05 10:47:33

   This program runs cyclically (default 100ms) and has access to all
   data points of the associated IEC 61850 device. Users can add custom
   logic in the designated sections below.
   ======================================================================== *)

PROGRAM PRG_GPS01GPC02UPM01FCB01
VAR
    (* ====== System Variables ====== *)
    cycle_count: UDINT := 0;           (* Increments each scan cycle *)
    first_scan: BOOL := TRUE;          (* TRUE only on first execution *)
    scan_time_ms: REAL := 0.0;         (* Last scan time in milliseconds *)

    (* ====== IED Connection Status ====== *)
    ied_connected: BOOL := FALSE;      (* TRUE when IED server is running *)
    ied_name: STRING := 'GPS01GPC02UPM01FCB01';
    device_name: STRING := 'GPS01GPC02UPM01FCB01';

    (* ====== Logical Devices ====== *)
    (* Available LDs: AnUn_ArcProtInput1, Application, BinIO, BinIO_BinaryInputs, BinIO_BinaryOutputs, CB1, CB1_Fundamental, Ds1, Ds2, Mod1, Mod1_Channel1, Mod2, Mod2_Channel1, Mod3, Mod3_Channel1, PowS, PowS_MeasPointI3ph1, PowS_MeasPointV3ph1, Rec, Rec_FaultRecorder, VI3p1, VI3p1_5051NOCgndB1, VI3p1_5051OC3phase1, VI3p1_ArcProtection1, VI3p1_Energy, VI3p1_FundSymComp, VI3p1_OperationalValues, VI3p1_ProcessMonitor, VI3p1_ExternalTrip1, VI3p1_67DirOC3phB1, VI3p1_67NDirOCgndB1, ComSupervision, ComSupervision_GOOSE *)

    (* ====== User Variables ====== *)
    (* Add your custom variables here *)
    (* Example:
    timer1: TON;
    counter: INT := 0;
    status_word: WORD;
    *)

END_VAR

(* ======================================================================
   INITIALIZATION SECTION
   Runs once on first scan. Use for setup and initialization.
   ====================================================================== *)
IF first_scan THEN
    (* Initialize user variables here *)
    cycle_count := 0;

    (* Log program start *)
    (* SCADA_LOG('INFO', CONCAT('PLC Program started: ', device_name)); *)

    first_scan := FALSE;
END_IF;

(* ======================================================================
   MAIN CYCLIC EXECUTION
   This section runs continuously every scan cycle (default 100ms).
   ====================================================================== *)

(* Increment cycle counter *)
cycle_count := cycle_count + 1;

(* ====== USER LOGIC SECTION 1: Pre-Processing ====== *)
(* Add logic that should run before main processing *)
(* Example:
IF ied_connected THEN
    (* Read IED data points *)
    (* status_word := READ_IED_DATA(device_name, 'LD0/MMXU1$MX$TotW$mag'); *)
END_IF;
*)

(* ====== USER LOGIC SECTION 2: Main Processing ====== *)
(* Add your main control logic here *)
(* Example:
IF counter > 100 THEN
    counter := 0;
    (* Perform periodic action *)
END_IF;
counter := counter + 1;
*)

(* ====== USER LOGIC SECTION 3: Post-Processing ====== *)
(* Add logic for outputs, writes, and cleanup *)
(* Example:
IF ied_connected THEN
    (* Write control commands to IED *)
    (* WRITE_IED_CONTROL(device_name, 'LD0/CSWI1$CO$Pos', TRUE); *)
END_IF;
*)

(* ====== Built-in Functions Available ====== *)
(*
   READ_IED_DATA(device: STRING, ref: STRING): ANY
       - Read data from IED object reference
       - Example: READ_IED_DATA('MyIED', 'LD0/MMXU1$MX$TotW$mag')

   WRITE_IED_DATA(device: STRING, ref: STRING, value: ANY): BOOL
       - Write data to IED object reference
       - Returns TRUE on success

   WRITE_IED_CONTROL(device: STRING, ref: STRING, value: ANY): BOOL
       - Send control command to IED
       - Returns TRUE on success

   SCADA_LOG(level: STRING, message: STRING)
       - Log message to event log
       - Levels: 'INFO', 'WARNING', 'ERROR'

   GET_DEVICE_STATUS(device: STRING): BOOL
       - Check if device is connected
*)

END_PROGRAM
